# B&R Automation Studio project MotionTestBenchMaster (part 24)

#### MNM.sfc - Cyclic code
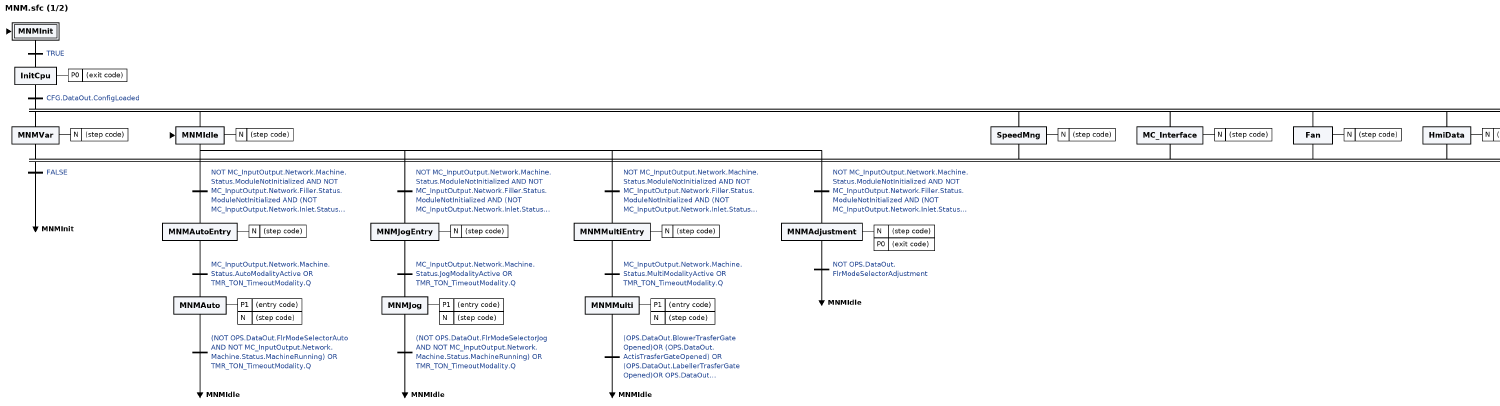
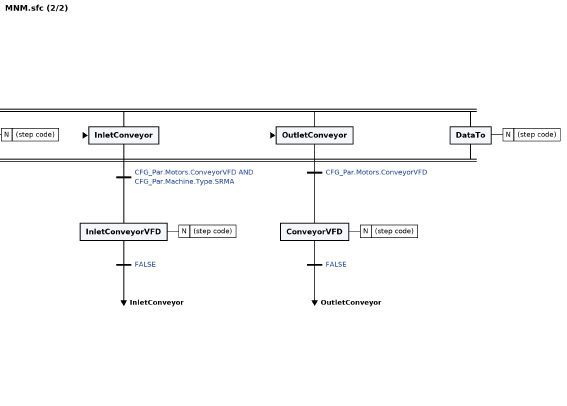
```iecst
PROGRAM _CYCLIC
INITIAL_STEP MNMInit:
END_STEP
TRANSITION FROM MNMInit TO InitCpu:=
TRUE
END_TRANSITION
STEP InitCpu:
END_STEP
EXIT_ACTION
InletConveyor_Hardware_CFG;
OutletConveyor_Hardware_CFG;
HMI_MNM_FlrSpeedWidget.AutoSpeedReq := REAL_TO_DINT(HMI_MNM_MinMachineSpeed);

HMI_CFG_PAR_1._020	:= TRUE;
HMI_CFG_PAR_1._160	:= _InCvrFC280.IN_ConfigPresent;//V 200.2.0
HMI_CFG_PAR_1._162	:= _OutCvrFC280.IN_ConfigPresent;

HMI_CFG_PAM_1._001	:= TRUE;//V 200.2.0
HMI_CFG_PAM_1._003	:= TRUE;
HMI_CFG_PAM_1._010	:= TRUE;
HMI_CFG_PAM_1._011	:= TRUE;
HMI_CFG_PAM_1._012	:= TRUE;
HMI_CFG_PAM_1._013	:= TRUE;
HMI_CFG_PAM_1._020	:= TRUE;

HMI_CFG_PAM_1._396	:= CFG_Par.Machine.Type.SRMA;//V 200.2.0
HMI_CFG_PAM_1._397	:= CFG_Par.Machine.Type.SRMA;//V 200.2.0
HMI_CFG_PAM_1._398	:= CFG_Par.Machine.Type.SRMA;//V 200.2.0
HMI_CFG_PAM_1._399	:= CFG_Par.Machine.Type.SRMA;//V 200.2.0
HMI_CFG_PAM_1._400	:= CFG_Par.Machine.Type.SRMA;//V 200.2.0
HMI_CFG_PAM_1._401	:= CFG_Par.Machine.Type.SRMA;//V 200.2.0
HMI_CFG_PAM_1._402	:= CFG_Par.Machine.Type.SRMA;//V 200.2.0
HMI_CFG_PAM_1._403	:= CFG_Par.Machine.Type.SRMA;//V 200.2.0
HMI_CFG_PAM_1._404	:= CFG_Par.ClosingUnit.Capper.Present;
HMI_CFG_PAM_1._405	:= CFG_Par.ClosingUnit.Capper.Present;
HMI_CFG_PAM_1._406	:= CFG_Par.ClosingUnit.Capper.Present;
HMI_CFG_PAM_1._407	:= CFG_Par.ClosingUnit.Capper.Present;
HMI_CFG_PAM_1._408	:= CFG_Par.ClosingUnit.Capper.Present;
HMI_CFG_PAM_1._409	:= CFG_Par.ClosingUnit.Capper.Present;
HMI_CFG_PAM_1._410	:= CFG_Par.ClosingUnit.Capper.Present;
HMI_CFG_PAM_1._411	:= CFG_Par.ClosingUnit.Capper.Present;
HMI_CFG_PAM_1._412	:= CFG_Par.Rinser.NoBottleNoSpray;//V 200.2.0
HMI_CFG_PAM_1._413	:= CFG_Par.Rinser.NoBottleNoSpray;//V 200.2.0
HMI_CFG_PAM_1._414	:= CFG_Par.Rinser.NoBottleNoSpray;//V 200.2.0
HMI_CFG_PAM_1._415	:= CFG_Par.Rinser.NoBottleNoSpray;//V 200.2.0
HMI_CFG_PAM_1._416	:= TRUE;//V 200.2.0
HMI_CFG_PAM_1._417	:= TRUE;//V 200.2.0
HMI_CFG_PAM_1._418	:= TRUE;//V 200.2.0
HMI_CFG_PAM_1._419	:= TRUE;//V 200.2.0
HMI_CFG_PAM_1._420	:= CFG_Par.ClosingUnit.Crowner.Present;
HMI_CFG_PAM_1._421	:= CFG_Par.ClosingUnit.Crowner.Present;
HMI_CFG_PAM_1._422	:= CFG_Par.ClosingUnit.Crowner.Present;
HMI_CFG_PAM_1._423	:= CFG_Par.ClosingUnit.Crowner.Present;
HMI_CFG_PAM_1._424	:= TRUE;
HMI_CFG_PAM_1._425	:= TRUE;
HMI_CFG_PAM_1._426	:= TRUE;
HMI_CFG_PAM_1._427	:= TRUE;
HMI_CFG_PAM_1._428	:= CFG_Par.FCI.Filltec OR CFG_Par.FCI.FTSystem OR CFG_Par.FCI.Heuft OR CFG_Par.FCI.Pressco OR CFG_Par.FCI.SIS OR CFG_Par.FCI.Stratec;//V4.A.A.1.7.0
HMI_CFG_PAM_1._429	:= CFG_Par.FCI.Filltec OR CFG_Par.FCI.FTSystem OR CFG_Par.FCI.Heuft OR CFG_Par.FCI.Pressco OR CFG_Par.FCI.SIS OR CFG_Par.FCI.Stratec;//V4.A.A.1.7.0
HMI_CFG_PAM_1._430	:= CFG_Par.FCI.Filltec OR CFG_Par.FCI.FTSystem OR CFG_Par.FCI.Heuft OR CFG_Par.FCI.Pressco OR CFG_Par.FCI.SIS OR CFG_Par.FCI.Stratec;//V4.A.A.1.7.0
HMI_CFG_PAM_1._431	:= CFG_Par.FCI.Filltec OR CFG_Par.FCI.FTSystem OR CFG_Par.FCI.Heuft OR CFG_Par.FCI.Pressco OR CFG_Par.FCI.SIS OR CFG_Par.FCI.Stratec;//V4.A.A.1.7.0
HMI_CFG_PAM_1._432	:= CFG_Par.FCI.Heuft OR CFG_Par.FCI.Stratec;
HMI_CFG_PAM_1._433	:= CFG_Par.FCI.Heuft OR CFG_Par.FCI.Stratec;
HMI_CFG_PAM_1._434	:= CFG_Par.FCI.Heuft OR CFG_Par.FCI.Stratec;
HMI_CFG_PAM_1._435	:= CFG_Par.FCI.Heuft OR CFG_Par.FCI.Stratec;
HMI_CFG_PAM_1._436	:= CFG_Par.Doser.Present; //v999hema
HMI_CFG_PAM_1._437	:= CFG_Par.Doser.Present; //v999hema
HMI_CFG_PAM_1._438	:= CFG_Par.Doser.Present; //v999hema
HMI_CFG_PAM_1._439	:= CFG_Par.Doser.Present; //v999hema

HMI_CFG_PAC_1._130	:= CFG_Par.Motors.FootbarPresent;
HMI_CFG_PAC_1._134  := CFG_Par.Machine.Type.SRMA AND CFG_Par.Lifting.Movements.Capper.UncoupledHeight > 0.0;//Capper Position For lifting movement
HMI_CFG_PAC_1._132	:= CFG_Par.Machine.Type.SRMA;
HMI_CFG_PAC_1._219	:= CFG_Par.Rinser.FootbarPresent;
HMI_CFG_PAC_1._220	:= CFG_Par.Rinser.FootbarPresent;
END_ACTION
TRANSITION FROM InitCpu TO (MNMVar,MNMIdle,SpeedMng,MC_Interface,Fan,HmiData,InletConveyor,OutletConveyor,DataTo):=
CFG.DataOut.ConfigLoaded
END_TRANSITION
STEP MNMVar:

VAR_MNM_NormalStop				:= AID.DataOut.ALR.Bit.ALR_MS_NormalStop;
VAR_MNM_QuickStop				:= AID.DataOut.ALR.Bit.ALR_MS_QuickStop;
VAR_MNM_NormalStopWithJog		:= AID.DataOut.ALR.Bit.ALR_MS_NormalWithJog;
VAR_MNM_NormalWithJogMnt		:= AID.DataOut.ALR.Bit.ALR_MS_NormalWithJogMnt; //V4.A.A.1.6.13
VAR_MNM_QuickStopWithJog		:= AID.DataOut.ALR.Bit.ALR_MS_QuickWithJog;
VAR_MNM_StopAfterEmpty 			:= AID.DataOut.ALR.Bit.ALR_CSR_StopAfterEmptying AND SFT.DataOut.MachineEmpty;//V 200.2.0

IF (MC_InputOutput.Network.Machine.Status.AutoModalityActive OR MC_InputOutput.Network.Machine.Status.MultiModalityActive) AND
	NOT VAR_MNM_NormalStop AND NOT VAR_MNM_QuickStop AND
	NOT VAR_MNM_NormalStopWithJog AND NOT  VAR_MNM_QuickStopWithJog AND NOT VAR_MNM_StopAfterEmpty THEN
	//added condition for stopping after pre-closing and washing cycle end//MasterBottle
	IF EDGEPOS(MAU_DumCon.DataOut.MachineStop) OR  EDGEPOS(SEL(CFG_Par.Process.BlendFill, SkdFlr.MachineStop, CrbFlr.MachineStop)) OR SFT.DataOut.FillingValvePositionReq OR CSR.DataOut.MachineStop OR EDGEPOS(CAP.DataOut.MachineStop) OR EDGEPOS(COP.DataOut.MachineStop) OR EDGEPOS(DOS.DataOut.MachineStop) OR EDGEPOS(RNS.DataOut.MachineStop) THEN//v999hema
		VAR_MNM_AutoStopRequest		:= TRUE;
		VAR_MNM_FlrAutoStopRequest	:= TRUE;
	END_IF

	IF (EDGEPOS(MAU_DumCon.DataOut.MachineStart) OR EDGEPOS(RNS.DataOut.MachineStart) OR EDGEPOS(SEL(CFG_Par.Process.BlendFill, SkdFlr.MachineStart, CrbFlr.MachineStart)) OR EDGEPOS(CAP.DataOut.MachineStart) OR EDGEPOS(COP.DataOut.MachineStart) OR EDGEPOS(DOS.DataOut.MachineStart) OR EDGEPOS(CRW.DataOut.MachineStart))
		AND NOT MAU_DumCon.DataOut.FillerReversePosReq AND NOT MAU_DumCon.DataOut.FillerFirstHalfPosReq AND NOT MAU_DumCon.DataOut.FillerSecondHalfPosReq THEN
		VAR_MNM_AutoStartRequest	:= TRUE;
		VAR_MNM_FlrAutoStartRequest := TRUE;
	END_IF
ELSE
	VAR_MNM_AutoStopRequest		:= FALSE;
	VAR_MNM_FlrAutoStopRequest	:= FALSE;
	VAR_MNM_AutoStartRequest	:= FALSE;
	VAR_MNM_FlrAutoStartRequest	:= FALSE;
END_IF

IF MC_InputOutput.Network.Machine.Status.AutoModalityActive THEN
	IF MC_InputOutput.Network.Machine.Status.MachineRunning THEN
		VAR_MNM_AutoStartRequest := FALSE;
	ELSE
		VAR_MNM_AutoStopRequest	:= FALSE;
	END_IF
	VAR_MNM_FlrAutoStopRequest	:= FALSE;
	VAR_MNM_FlrAutoStartRequest	:= FALSE;
ELSIF MC_InputOutput.Network.Machine.Status.MultiModalityActive THEN
	IF MC_InputOutput.Network.Filler.Status.ModuleRunning THEN
		VAR_MNM_FlrAutoStartRequest	:= FALSE;
	ELSE
		VAR_MNM_FlrAutoStopRequest	:= FALSE;
	END_IF
	VAR_MNM_AutoStopRequest		:= FALSE;
	VAR_MNM_AutoStartRequest	:= FALSE;
END_IF

(* Machine Start and Stop Management *)
VAR_MNM_FpMachineStartPb := EDGEPOS(HMI_CmdBar_PB[PB_FillerStartStop].Command);

//V4 200.2.0
VAR_MNM_MachineStart	:= IO_PB_FlStart.ON AND IO_PB_FlStart.Enable;
VAR_MNM_MachineStop		:= IO_PB_FlStop.ON;
END_STEP
STEP MNMIdle:
VAR_MNM_HornFlrRequest				:= FALSE;

MNM.DataOut.StartLightFixRequest	:= FALSE;
MNM.DataOut.StartLightBlinkRequest	:= FALSE;

TMR_TON_StartingHornElapsed.IN		:= FALSE;

TMR_TON_TimeoutModality.IN			:= FALSE;
TMR_TON_TimeoutModality();

FlrFmc.FillerOneStepReceived		:= FALSE;

MC_InputOutput.Network.Machine.Commands.MachineStart				:= FALSE;
MC_InputOutput.Network.Machine.Commands.JogPushButton				:= FALSE;
MC_InputOutput.Network.Machine.Commands.StepByStepModalityRequest	:= FALSE;
MC_InputOutput.Network.Machine.Commands.InMotionTimerModReq			:= FALSE;
MC_InputOutput.Network.Machine.Commands.StepByStepSingleAxisModReq	:= FALSE;//V1.7.2
MC_InputOutput.Network.Machine.Commands.PositioningModalityRequest	:= FALSE;//V1.7.2

MC_InputOutput.Network.Machine.Commands.AutoModalityRequest			:= FALSE;
MC_InputOutput.Network.Machine.Commands.AutoCombiModalityRequest	:= FALSE;
MC_InputOutput.Network.Machine.Commands.JogMachineModalityRequest	:= FALSE;
MC_InputOutput.Network.Machine.Commands.MultiModalityRequest		:= FALSE;

MC_InputOutput.Network.Filler.Commands.AutoFillerModule				:= FALSE;
MC_InputOutput.Network.Filler.Commands.JogFillerModule				:= FALSE;
MC_InputOutput.Network.Filler.Commands.StartFillerModule			:= FALSE;
MC_InputOutput.Network.Filler.Commands.JogPushButtonFillerModule	:= FALSE;

MC_InputOutput.Network.Inlet.Commands.AutoInletModule				:= FALSE;
MC_InputOutput.Network.Inlet.Commands.JogInletModule				:= FALSE;
MC_InputOutput.Network.Inlet.Commands.StartInletModule				:= FALSE;
MC_InputOutput.Network.Inlet.Commands.JogPushButtonInletModule		:= FALSE;

MC_InputOutput.Network.Outlet.Commands.AutoOutletModule				:= FALSE;
MC_InputOutput.Network.Outlet.Commands.JogOutletModule				:= FALSE;
MC_InputOutput.Network.Outlet.Commands.StartOutletModule			:= FALSE;
MC_InputOutput.Network.Outlet.Commands.JogPushButtonOutletModule	:= FALSE;
END_STEP
TRANSITION AutoMode FROM MNMIdle TO MNMAutoEntry:=
NOT MC_InputOutput.Network.Machine.Status.ModuleNotInitialized AND//v1.7.2a
NOT MC_InputOutput.Network.Filler.Status.ModuleNotInitialized AND//VXXXXXX
(NOT MC_InputOutput.Network.Inlet.Status.ModuleNotInitialized	OR MC_InputOutput.Network.Inlet.Status.ModuleReal)	AND
(NOT MC_InputOutput.Network.Outlet.Status.ModuleNotInitialized	OR MC_InputOutput.Network.Outlet.Status.ModuleReal)	AND
MC_InputOutput.Network.Machine.Status.EnableAuto				AND
OPS.DataOut.FlrModeSelectorAuto		AND //V4 200.2.0
NOT MC_InputOutput.Network.Machine.Exceptions.DcBusLowMachineException//V4.A.A.1.7.0
END_TRANSITION
TRANSITION JogMode FROM MNMIdle TO MNMJogEntry:=
NOT MC_InputOutput.Network.Machine.Status.ModuleNotInitialized AND//v1.7.2a
NOT MC_InputOutput.Network.Filler.Status.ModuleNotInitialized	AND
(NOT MC_InputOutput.Network.Inlet.Status.ModuleNotInitialized	OR MC_InputOutput.Network.Inlet.Status.ModuleReal)	AND
(NOT MC_InputOutput.Network.Outlet.Status.ModuleNotInitialized	OR MC_InputOutput.Network.Outlet.Status.ModuleReal)	AND
MC_InputOutput.Network.Machine.Status.EnableJog					AND
OPS.DataOut.FlrModeSelectorJog	AND
NOT MC_InputOutput.Network.Machine.Exceptions.DcBusLowMachineException//V4 200.2.0
END_TRANSITION
STEP MNMJogEntry:
MC_InputOutput.Network.Machine.Commands.JogMachineModalityRequest		:= TRUE;
TMR_TON_TimeoutModality(IN := TRUE, PT := t#2s);
END_STEP
TRANSITION JogModeActive FROM MNMJogEntry TO MNMJog:=
MC_InputOutput.Network.Machine.Status.JogModalityActive OR TMR_TON_TimeoutModality.Q
END_TRANSITION
STEP MNMJog:
MC_InputOutput.Network.Machine.Commands.JogMachineModalityRequest		:= TRUE;

IF VAR_MNM_NormalStop OR VAR_MNM_QuickStop THEN
	VAR_MNM_JogStep := MNM_JogFault;
ELSIF NOT (NOT MC_InputOutput.Network.Machine.Status.NoModalityActive AND MC_InputOutput.Network.Machine.Status.JogModalityActive) THEN
	VAR_MNM_JogStep := MNM_JogWaitStart;
ELSIF EDGENEG(OPS.DataOut.JogStartPb)  THEN
	VAR_MNM_JogStep := MNM_JogWaitStart;
END_IF

TMR_TON_StartingHornElapsed.IN	:= FALSE;
MC_InputOutput.Network.Machine.Commands.JogPushButton				:= FALSE;
VAR_MNM_HornFlrRequest	:= FALSE;

CASE VAR_MNM_JogStep OF
	MNM_JogWaitStart:
		IF OPS.DataOut.JogStartPb AND NOT CSR.DataOut.MachineStop THEN (*Master nuovo*)
			VAR_MNM_JogStep := MNM_JogHornBlow;
		END_IF

	MNM_JogHornBlow:
		TMR_TON_StartingHornElapsed.IN	:= TRUE;
		VAR_MNM_HornFlrRequest	:= TRUE;

		IF TMR_TON_StartingHornElapsed.Q THEN
			VAR_MNM_JogStep := MNM_JogMachineStart;
		END_IF

	MNM_JogMachineStart:
		MC_InputOutput.Network.Machine.Commands.JogPushButton := TRUE;

		IF MC_InputOutput.Network.Machine.Status.MachineRunning THEN
			VAR_MNM_JogStep := MNM_JogMachineRunning;
		END_IF

	MNM_JogMachineRunning:
		MC_InputOutput.Network.Machine.Commands.JogPushButton := TRUE;

	MNM_JogMachineStopping:
		IF NOT MC_InputOutput.Network.Machine.Status.MachineRunning THEN
			VAR_MNM_JogStep := MNM_JogWaitStart;
		END_IF

	MNM_JogFault:
		IF NOT VAR_MNM_NormalStop AND NOT VAR_MNM_QuickStop THEN
			VAR_MNM_JogStep := MNM_JogWaitStart;
		END_IF
END_CASE

TMR_TON_StartingHornElapsed(PT:= t#2s);
END_STEP
ENTRY_ACTION
VAR_MNM_JogStep := MNM_JogWaitStart;
END_ACTION
TRANSITION IdleMode FROM MNMJog TO MNMIdle:=
(NOT OPS.DataOut.FlrModeSelectorJog AND NOT MC_InputOutput.Network.Machine.Status.MachineRunning) OR //V 200.2.0
TMR_TON_TimeoutModality.Q
END_TRANSITION
(* @SFCISJUMP := 'MNMIdle' *)
TRANSITION MultiMode FROM MNMIdle TO MNMMultiEntry:=
NOT MC_InputOutput.Network.Machine.Status.ModuleNotInitialized AND
NOT MC_InputOutput.Network.Filler.Status.ModuleNotInitialized	AND
(NOT MC_InputOutput.Network.Inlet.Status.ModuleNotInitialized	OR MC_InputOutput.Network.Inlet.Status.ModuleReal)	AND
(NOT MC_InputOutput.Network.Outlet.Status.ModuleNotInitialized	OR MC_InputOutput.Network.Outlet.Status.ModuleReal)	AND
NOT OPS.DataOut.FlrModeSelectorAdjustment	AND
MC_InputOutput.Network.Machine.Status.EnableMulti	AND
NOT (OPS.DataOut.BlowerTrasferGateOpened AND OPS.DataOut.ActisTrasferGateOpened)AND //da cambiare
NOT MC_InputOutput.Network.Machine.Exceptions.DcBusLowMachineException
END_TRANSITION
STEP MNMMultiEntry:
MC_InputOutput.Network.Machine.Commands.MultiModalityRequest	:= TRUE;
TMR_TON_TimeoutModality(IN := TRUE, PT := t#2s);
END_STEP
TRANSITION MultiModeActive FROM MNMMultiEntry TO MNMMulti:=
MC_InputOutput.Network.Machine.Status.MultiModalityActive OR TMR_TON_TimeoutModality.Q
END_TRANSITION
STEP MNMMulti:
MC_InputOutput.Network.Machine.Commands.MultiModalityRequest	:= TRUE;

(* FILLER MULTI *)
IF EDGE(OPS.DataOut.FlrModeSelectorAuto) THEN
	VAR_MNM_FlrMultiStep := MNM_MultiModeSelection;
ELSIF VAR_MNM_FlrMultiStep >= MNM_MultiAutoWaitStart AND VAR_MNM_FlrMultiStep <= MNM_MultiAutoMachineStopping THEN
	IF VAR_MNM_NormalStop OR VAR_MNM_QuickStop OR VAR_MNM_NormalStopWithJog OR VAR_MNM_QuickStopWithJog OR VAR_MNM_StopAfterEmpty OR VAR_MNM_StopIfNotEmpty THEN
		VAR_MNM_FlrMultiStep := MNM_MultiFault;
	ELSIF NOT VAR_MNM_MachineStop OR VAR_MNM_FlrAutoStopRequest THEN
		VAR_MNM_FlrMultiStep := MNM_MultiAutoMachineStopping;
	END_IF
ELSIF VAR_MNM_FlrMultiStep >= MNM_MultiJogWaitStart AND VAR_MNM_FlrMultiStep <= MNM_MultiJogMachineStopping THEN
	IF VAR_MNM_NormalStop OR VAR_MNM_QuickStop THEN
		VAR_MNM_FlrMultiStep := MNM_MultiFault;
	ELSIF EDGENEG(OPS.DataOut.JogStartPb)  THEN
		VAR_MNM_FlrMultiStep := MNM_MultiJogMachineStopping;
	END_IF
END_IF

TMR_TON_StartingHornElapsed.IN	:= FALSE;
MC_InputOutput.Network.Filler.Commands.AutoFillerModule				:= FALSE;
MC_InputOutput.Network.Filler.Commands.StartFillerModule			:= FALSE;
MC_InputOutput.Network.Filler.Commands.JogFillerModule				:= FALSE;
MC_InputOutput.Network.Filler.Commands.JogPushButtonFillerModule	:= FALSE;
VAR_MNM_HornFlrRequest					:= FALSE;
MNM.DataOut.StartLightFixRequest		:= FALSE;
MNM.DataOut.StartLightBlinkRequest		:= FALSE;

CASE VAR_MNM_FlrMultiStep OF
	MNM_MultiModeSelection:
		IF OPS.DataOut.FlrModeSelectorAuto AND MC_InputOutput.Network.Filler.Status.EnableAutoModality THEN
			VAR_MNM_FlrMultiStep := MNM_MultiAutoWaitStart;
		ELSIF OPS.DataOut.FlrModeSelectorJog AND MC_InputOutput.Network.Filler.Status.EnableJogModality THEN
			VAR_MNM_FlrMultiStep := MNM_MultiJogWaitStart;
		END_IF

	MNM_MultiAutoWaitStart:
		MC_InputOutput.Network.Filler.Commands.AutoFillerModule := TRUE;
		MNM.DataOut.StartLightBlinkRequest	:= TRUE;

		IF ((VAR_MNM_MachineStart OR VAR_MNM_FlrAutoStartRequest) AND VAR_MNM_MachineStop AND MC_InputOutput.Network.Filler.Status.EnableAutoModality) THEN
			VAR_MNM_FlrMultiStep	:= MNM_MultiAutoHornBlow;
		ELSIF VAR_MNM_AutoVortexCalibActive THEN
			VAR_MNM_FlrMultiStep	:= MNM_MultiVortexCalibIdle;
		ELSIF FmcFlr.VortexCalibrActive THEN
			VAR_MNM_FlrMultiStep 	:= MNM_MultiVortexCalibHornBlow;
		ELSIF HMI_MNM_PB[PB_MNM_AxisStepByStep].ON THEN
			VAR_MNM_FlrMultiStep 	:= MNM_MultiStepHornBlow;
		ELSIF HMI_MNM_PB[PB_MNM_FootboardPosition].ON THEN
			VAR_MNM_FlrMultiStep 	:= MNM_MultiFootboardHornBlow;
		ELSIF CAP.DataOut.GreasingPositioningReq OR CSR.DataOut.CapPositioningReq THEN//V4.A.A.1.7.0
			VAR_MNM_FlrMultiStep	:= MNM_MultiCapperPosHornBlow;
		END_IF

	MNM_MultiAutoHornBlow:
		MC_InputOutput.Network.Filler.Commands.AutoFillerModule	:= TRUE;
		MNM.DataOut.StartLightFixRequest	:= TRUE;
		TMR_TON_StartingHornElapsed.IN		:= TRUE;
		VAR_MNM_HornFlrRequest	:= TRUE;

		IF NOT ((VAR_MNM_MachineStart OR VAR_MNM_FlrAutoStartRequest) AND VAR_MNM_MachineStop AND MC_InputOutput.Network.Filler.Status.EnableAutoModality) THEN
			VAR_MNM_FlrMultiStep := MNM_MultiAutoWaitStart;
		END_IF

		IF TMR_TON_StartingHornElapsed.Q THEN
			VAR_MNM_FlrMultiStep := MNM_MultiAutoMachineStart;
		END_IF

	MNM_MultiAutoMachineStart:
		MC_InputOutput.Network.Filler.Commands.AutoFillerModule		:= TRUE;
		MC_InputOutput.Network.Filler.Commands.StartFillerModule	:= TRUE;
		MNM.DataOut.StartLightFixRequest	:= TRUE;

		IF MC_InputOutput.Network.Filler.Status.ModuleRunning THEN
			VAR_MNM_FlrMultiStep := MNM_MultiAutoMachineRunning;
		END_IF

	MNM_MultiAutoMachineRunning:	//Wait stop PB or Fault
		MC_InputOutput.Network.Filler.Commands.AutoFillerModule		:= TRUE;
		MC_InputOutput.Network.Filler.Commands.StartFillerModule	:= TRUE;
		MNM.DataOut.StartLightFixRequest	:= TRUE;

	MNM_MultiAutoMachineStopping:
		MC_InputOutput.Network.Filler.Commands.AutoFillerModule		:= TRUE;

		IF NOT MC_InputOutput.Network.Filler.Status.ModuleRunning THEN
			VAR_MNM_FlrMultiStep := MNM_MultiAutoWaitStart;
		END_IF

	MNM_MultiVortexCalibHornBlow:
		TMR_TON_StartingHornElapsed.IN	:= TRUE;
		VAR_MNM_HornFlrRequest	:= TRUE;

		IF TMR_TON_StartingHornElapsed.Q THEN
			VAR_MNM_FlrMultiStep := MNM_MultiVortexCalibPosStart;
		END_IF

	MNM_MultiVortexCalibPosStart:
		MC_InputOutput.Network.Filler.Parameters.StepNumber	:= 1;
		MC_InputOutput.Network.Filler.Commands.StepByStepModalityRequest	:= TRUE;

		IF MC_InputOutput.Network.Filler.Status.StepByStepModalityActive THEN
			VAR_MNM_FlrMultiStep := MNM_MultiVortexCalibPosWaitStop;
		END_IF

	MNM_MultiVortexCalibPosWaitStop:
		IF NOT MC_InputOutput.Network.Filler.Status.StepByStepModalityActive AND NOT MC_InputOutput.Network.Filler.Status.ModuleRunning THEN
			VAR_MNM_FlrMultiStep := MNM_MultiVortexCalibIdle;
			VAR_MNM_AutoVortexCalibActive := TRUE;
		END_IF

	MNM_MultiVortexCalibIdle:
		IF EDGEPOS(FmcFlr.FillerOneStepReq) THEN
			VAR_MNM_FlrMultiStep := MNM_MultiStepFmcHornBlow;
		END_IF

		IF NOT FmcFlr.VortexCalibrActive THEN
			VAR_MNM_AutoVortexCalibActive := FALSE;
			VAR_MNM_FlrMultiStep := MNM_MultiAutoWaitStart;
		END_IF

	MNM_MultiStepFmcHornBlow:
		TMR_TON_StartingHornElapsed.IN	:= TRUE;
		VAR_MNM_HornFlrRequest	:= TRUE;

		IF TMR_TON_StartingHornElapsed.Q THEN
			FlrFmc.FillerOneStepReceived	:= FmcFlr.FillerOneStepReq;
			VAR_MNM_FlrMultiStep := MNM_MultiStepFmcStart;
		END_IF

	MNM_MultiStepFmcStart:
		MC_InputOutput.Network.Filler.Parameters.StepNumber	:= 1;
		MC_InputOutput.Network.Filler.Commands.StepByStepModalityRequest	:= TRUE;

		IF MC_InputOutput.Network.Filler.Status.StepByStepModalityActive THEN
			VAR_MNM_FlrMultiStep := MNM_MultiStepFmcWaitStop;
		END_IF

	MNM_MultiStepFmcWaitStop:
		IF NOT MC_InputOutput.Network.Filler.Status.StepByStepModalityActive AND NOT MC_InputOutput.Network.Filler.Status.ModuleRunning THEN
			VAR_MNM_FlrMultiStep := MNM_MultiVortexCalibIdle;
		END_IF

	MNM_MultiStepHornBlow:
		TMR_TON_StartingHornElapsed.IN	:= TRUE;
		VAR_MNM_HornFlrRequest	:= TRUE;

		IF TMR_TON_StartingHornElapsed.Q THEN
			VAR_MNM_FlrMultiStep := MNM_MultiStepStart;
		END_IF

	MNM_MultiStepStart:
		MC_InputOutput.Network.Filler.Parameters.StepNumber	:= HMI_MNM_AxisStepByStepOffset;
		MC_InputOutput.Network.Filler.Commands.StepByStepModalityRequest	:= TRUE;

		IF MC_InputOutput.Network.Filler.Status.StepByStepModalityActive THEN
			VAR_MNM_FlrMultiStep := MNM_MultiStepWaitStop;
		END_IF

	MNM_MultiStepWaitStop:
		IF NOT MC_InputOutput.Network.Filler.Status.StepByStepModalityActive AND NOT MC_InputOutput.Network.Filler.Status.ModuleRunning THEN
			VAR_MNM_FlrMultiStep := MNM_MultiAutoWaitStart;
		END_IF

	MNM_MultiFootboardHornBlow:
		TMR_TON_StartingHornElapsed.IN	:= TRUE;
		VAR_MNM_HornFlrRequest	:= TRUE;

		IF TMR_TON_StartingHornElapsed.Q THEN
			VAR_MNM_FlrMultiStep := MNM_MultiFootboardStart;
		END_IF

	MNM_MultiFootboardStart:
		IF LREAL_TO_INT(MC_InputOutput.Network.Filler.Status.FillerAbsolutePosition / 360.0) < HMI_PAC_1._130 THEN
			MC_InputOutput.Network.Filler.Parameters.StepNumber		:= HMI_PAC_1._130 - (LREAL_TO_INT(MC_InputOutput.Network.Filler.Status.FillerAbsolutePosition / 360.0));
		ELSE
			MC_InputOutput.Network.Filler.Parameters.StepNumber	:= HMI_PAC_1._100 - (LREAL_TO_INT(MC_InputOutput.Network.Filler.Status.FillerAbsolutePosition / 360.0)) + HMI_PAC_1._130;
		END_IF

		MC_InputOutput.Network.Filler.Commands.StepByStepModalityRequest	:= TRUE;

		IF MC_InputOutput.Network.Filler.Status.StepByStepModalityActive THEN
			VAR_MNM_FlrMultiStep := MNM_MultiFootboardWaitStop;
		END_IF

	MNM_MultiFootboardWaitStop:
		IF NOT MC_InputOutput.Network.Filler.Status.StepByStepModalityActive AND NOT MC_InputOutput.Network.Filler.Status.ModuleRunning THEN
			VAR_MNM_FlrMultiStep := MNM_MultiAutoWaitStart;
		END_IF

	MNM_MultiCapperPosHornBlow:

	MNM_MultiCapperPosStart:

	MNM_MultiCapperPosWaitStop:

	MNM_MultiCapperFinePosStart:

	MNM_MultiCapperFinePosWaitStop:

	MNM_MultiJogWaitStart:
		MC_InputOutput.Network.Filler.Commands.JogFillerModule	:= TRUE;
		IF OPS.DataOut.JogStartPb THEN
			VAR_MNM_FlrMultiStep := MNM_MultiJogHornBlow;
		END_IF

	MNM_MultiJogHornBlow:
		MC_InputOutput.Network.Filler.Commands.JogFillerModule	:= TRUE;
		TMR_TON_StartingHornElapsed.IN	:= TRUE;
		VAR_MNM_HornFlrRequest	:= TRUE;

		IF TMR_TON_StartingHornElapsed.Q THEN
			VAR_MNM_FlrMultiStep := MNM_MultiJogMachineStart;
		END_IF

	MNM_MultiJogMachineStart:
		MC_InputOutput.Network.Filler.Commands.JogFillerModule	:= TRUE;
		MC_InputOutput.Network.Filler.Commands.JogPushButtonFillerModule := TRUE;

		IF MC_InputOutput.Network.Filler.Status.ModuleRunning THEN
			VAR_MNM_FlrMultiStep := MNM_MultiJogMachineRunning;
		END_IF

	MNM_MultiJogMachineRunning:
		MC_InputOutput.Network.Filler.Commands.JogFillerModule	:= TRUE;
		MC_InputOutput.Network.Filler.Commands.JogPushButtonFillerModule:= TRUE;

	MNM_MultiJogMachineStopping:
		MC_InputOutput.Network.Filler.Commands.JogFillerModule	:= TRUE;
		IF NOT MC_InputOutput.Network.Filler.Status.ModuleRunning THEN
			VAR_MNM_FlrMultiStep := MNM_MultiJogWaitStart;
		END_IF

	MNM_MultiFault:
		MC_InputOutput.Network.Filler.Commands.AutoFillerModule		:= OPS.DataOut.FlrModeSelectorAuto AND MC_InputOutput.Network.Filler.Status.EnableAutoModality;//V4.A.A.1.6.12d
		MC_InputOutput.Network.Filler.Commands.JogFillerModule		:= OPS.DataOut.FlrModeSelectorJog AND MC_InputOutput.Network.Filler.Status.EnableJogModality;//V4.A.A.1.6.12d

		IF NOT (VAR_MNM_NormalStop OR VAR_MNM_QuickStop OR VAR_MNM_NormalStopWithJog OR VAR_MNM_QuickStopWithJog OR VAR_MNM_StopAfterEmpty OR VAR_MNM_StopIfNotEmpty) THEN
			VAR_MNM_FlrMultiStep := MNM_MultiAutoWaitStart;//V4.A.A.1.6.12d
		ELSIF MC_InputOutput.Network.Filler.Status.ModuleJogActive THEN
			IF NOT VAR_MNM_NormalStop AND NOT VAR_MNM_QuickStop THEN
				VAR_MNM_FlrMultiStep := MNM_MultiJogWaitStart;
			END_IF
		END_IF
END_CASE

TMR_TON_StartingHornElapsed(PT:= t#2s);
END_STEP
ENTRY_ACTION
VAR_MNM_FlrMultiStep		:= MNM_MultiModeSelection;
VAR_MNM_FlrInletMultiStep	:= MNM_MultiModeSelection;
END_ACTION
TRANSITION IdleMode FROM MNMMulti TO MNMIdle:=
(OPS.DataOut.BlowerTrasferGateOpened)OR//da controllare in collaudo
(OPS.DataOut.ActisTrasferGateOpened) OR//da controllare in collaudo
(OPS.DataOut.LabellerTrasferGateOpened)OR//da controllare in collaudo
OPS.DataOut.FlrModeSelectorAdjustment OR TMR_TON_TimeoutModality.Q
END_TRANSITION
(* @SFCISJUMP := 'MNMIdle' *)
TRANSITION AdjustmentMode FROM MNMIdle TO MNMAdjustment:=
NOT MC_InputOutput.Network.Machine.Status.ModuleNotInitialized AND
NOT MC_InputOutput.Network.Filler.Status.ModuleNotInitialized	AND
(NOT MC_InputOutput.Network.Inlet.Status.ModuleNotInitialized	OR MC_InputOutput.Network.Inlet.Status.ModuleReal)	AND
(NOT MC_InputOutput.Network.Outlet.Status.ModuleNotInitialized	OR MC_InputOutput.Network.Outlet.Status.ModuleReal)	AND
OPS.DataOut.FlrModeSelectorAdjustment AND
NOT MC_InputOutput.Network.Machine.Exceptions.DcBusLowMachineException
END_TRANSITION
STEP MNMAdjustment:
IF VAR_MNM_NormalStop OR VAR_MNM_QuickStop OR VAR_MNM_NormalStopWithJog OR VAR_MNM_QuickStopWithJog OR VAR_MNM_StopAfterEmpty OR VAR_MNM_StopIfNotEmpty THEN//V4.A.A.1.7.0
	VAR_MNM_AdjustmentStep := MNM_AdjFault;
END_IF
IF EDGEPOS(HMI_MNM_PB[PB_MNM_AxisPositioning].ON) THEN
	MC_InputOutput.Network.Machine.Commands.PositioningModalityRequest	:=  TRUE;
ELSIF MC_InputOutput.Network.Machine.Status.PositioningModalityActive OR NOT HMI_MNM_PB[PB_MNM_AxisPositioning].ON THEN
	MC_InputOutput.Network.Machine.Commands.PositioningModalityRequest	:=  FALSE;
END_IF

IF EDGENEG(MC_InputOutput.Network.Machine.Status.PositioningModalityActive) THEN
	HMI_MNM_AxisPositionOffset	:= 0.0;
END_IF

IF EDGEPOS(HMI_MNM_PB[PB_MNM_AxisHoming].ON) THEN
	MC_InputOutput.Network.Machine.Commands.SelectiveHomeModalityRequest	:= TRUE;
ELSIF MC_InputOutput.Network.Machine.Status.SelectiveHomeModalityActive OR NOT HMI_MNM_PB[PB_MNM_AxisHoming].ON THEN
	MC_InputOutput.Network.Machine.Commands.SelectiveHomeModalityRequest	:= FALSE;
END_IF

MC_InputOutput.Network.Machine.Commands.BrakeReleaseModalityRequest	:= HMI_MNM_PB[PB_MNM_BrakeRelease].ON;

MC_InputOutput.Network.Machine.Commands.VelocityModalityRequest		:= HMI_MNM_PB[PB_MNM_VelocityTest].ON;
MC_InputOutput.Network.Machine.Parameters.ManualVelocity			:= REAL_TO_UINT(HMI_MNM_ConveyorSpeed / 10.0);

TMR_TON_StartingHornElapsed.IN	:= FALSE;
VAR_MNM_HornFlrRequest	:= FALSE;
MNM.DataOut.StartLightFixRequest	:= FALSE;
MNM.DataOut.StartLightBlinkRequest	:= FALSE;

CASE VAR_MNM_AdjustmentStep OF
	MNM_AdjWaitStart:
		VAR_MNM_AdjAxisPositionOffset := 0.0;

		//MNM.DataOut.StartLightBlinkRequest	:= TRUE; v4 200.2.0 // no blink PB start in Adjustment modality

		IF HMI_MNM_PB[PB_MNM_FootboardPosition].ON THEN
			VAR_MNM_AdjustmentStep := MNM_AdjFillerFootbarSettingPos;
		ELSIF  HMI_MNM_PB[PB_MNM_RinserFootboardPosition].ON THEN
			VAR_MNM_AdjustmentStep := MNM_AdjRinserFootbarSettingPos;
		ELSIF CAP.DataOut.GreasingPositioningReq  THEN
			VAR_MNM_AdjustmentStep := MNM_AdjCapGreasingSettingPos;
		ELSIF CSR.DataOut.CrwPositioningReq THEN
			VAR_MNM_AdjustmentStep := MNM_AdjCrownerSettingPos;
		ELSIF CSR.DataOut.CapPositioningReq THEN
			VAR_MNM_AdjustmentStep := MNM_AdjCapperSettingPos;
		END_IF
	//Filler Footbar
	MNM_AdjFillerFootbarSettingPos:

		VAR_MNM_AdjAxisFillerFootBar := TRUE;

		HMI_MNM_AxisSelected := CFG_MC.Mechanical.ReferenceId.Filler + CST_FillerSubModuleHmiStart;
		VAR_MNM_AdjAxisPositionOffset := 0.0;

		IF LREAL_TO_INT(MC_InputOutput.Network.Filler.Status.FillerAbsolutePosition / 360.0) < HMI_PAC_1._130 THEN
			MC_InputOutput.Network.Machine.Parameters.StepNumber		:= HMI_PAC_1._130 - (LREAL_TO_INT(MC_InputOutput.Network.Filler.Status.FillerAbsolutePosition / 360.0));
		ELSE
			MC_InputOutput.Network.Machine.Parameters.StepNumber	:= HMI_PAC_1._100 - (LREAL_TO_INT(MC_InputOutput.Network.Filler.Status.FillerAbsolutePosition / 360.0)) + HMI_PAC_1._130;
		END_IF

		VAR_MNM_AdjustmentStep := MNM_AdjHornBlow;
	//Rinser Footbar
	MNM_AdjRinserFootbarSettingPos:

		VAR_MNM_AdjAxisRinserFootBar	:= TRUE;

		HMI_MNM_AxisSelected := CFG_MC.Mechanical.ReferenceId.Rinser + CST_FillerSubModuleHmiStart;
		VAR_MNM_AdjAxisPositionOffset := 0.0;

		IF LREAL_TO_INT(MC_InputOutput.Network.Filler.Status.RinserAbsolutePosition / 360.0) < HMI_PAC_1._220 THEN
			MC_InputOutput.Network.Machine.Parameters.StepNumber		:= HMI_PAC_1._220 - (LREAL_TO_INT(MC_InputOutput.Network.Filler.Status.RinserAbsolutePosition / 360.0));
		ELSE
			MC_InputOutput.Network.Machine.Parameters.StepNumber	:= HMI_PAC_1._200- (LREAL_TO_INT(MC_InputOutput.Network.Filler.Status.RinserAbsolutePosition / 360.0)) + HMI_PAC_1._220;
		END_IF

		VAR_MNM_AdjustmentStep := MNM_AdjHornBlow;
	//Doser Pos
	MNM_AdjDoserFootbarSettingPos:

		HMI_MNM_AxisSelected := CFG_MC.Mechanical.ReferenceId.Rinser + CST_FillerSubModuleHmiStart;
		VAR_MNM_AdjAxisPositionOffset := 0.0;

		IF LREAL_TO_INT(MC_InputOutput.Network.Filler.Status.FillerAbsolutePosition / 360.0) < HMI_PAC_1._130 THEN//
			MC_InputOutput.Network.Machine.Parameters.StepNumber		:= HMI_PAC_1._130 - (LREAL_TO_INT(MC_InputOutput.Network.Filler.Status.FillerAbsolutePosition / 360.0));
		ELSE
			MC_InputOutput.Network.Machine.Parameters.StepNumber	:= HMI_PAC_1._500- (LREAL_TO_INT(MC_InputOutput.Network.Filler.Status.FillerAbsolutePosition / 360.0)) + HMI_PAC_1._130;
		END_IF

		VAR_MNM_AdjustmentStep := MNM_AdjHornBlow;
	//Capper pos For lifting
	MNM_AdjCapperSettingPos:

		HMI_MNM_AxisSelected := CFG_MC.Mechanical.ReferenceId.Capper + CST_FillerSubModuleHmiStart;
		VAR_MNM_AdjAxisPositionOffset := HMI_PAM_3._540;

		IF LREAL_TO_INT(MC_InputOutput.Network.Filler.Status.CapperAbsolutePosition / 360.0) < HMI_PAC_1._134 THEN
			MC_InputOutput.Network.Machine.Parameters.StepNumber		:= HMI_PAC_1._134 - (LREAL_TO_INT(MC_InputOutput.Network.Filler.Status.CapperAbsolutePosition / 360.0));//Fra
		ELSE
			MC_InputOutput.Network.Machine.Parameters.StepNumber	:= HMI_PAC_1._400 - (LREAL_TO_INT(MC_InputOutput.Network.Filler.Status.CapperAbsolutePosition / 360.0)) + HMI_PAC_1._134;//Fra
		END_IF

		VAR_MNM_AdjustmentStep := MNM_AdjHornBlow;

	//Crowner  Pos For Lifting
	MNM_AdjCrownerSettingPos:

		HMI_MNM_AxisSelected := CFG_MC.Mechanical.ReferenceId.Crowner + CST_FillerSubModuleHmiStart;
		VAR_MNM_AdjAxisPositionOffset := HMI_PAM_3._410;

		IF LREAL_TO_INT(MC_InputOutput.Network.Filler.Status.CrownerAbsolutePosition / 360.0) < HMI_PAC_1._133 THEN
			MC_InputOutput.Network.Machine.Parameters.StepNumber		:= HMI_PAC_1._133 - (LREAL_TO_INT(MC_InputOutput.Network.Filler.Status.CrownerAbsolutePosition / 360.0));//Fra
		ELSE
			MC_InputOutput.Network.Machine.Parameters.StepNumber	:= HMI_PAC_1._300 - (LREAL_TO_INT(MC_InputOutput.Network.Filler.Status.CrownerAbsolutePosition / 360.0)) + HMI_PAC_1._133;//Fra
		END_IF

		VAR_MNM_AdjustmentStep := MNM_AdjHornBlow;
	//Capper Greasing Pos
	MNM_AdjCapGreasingSettingPos:

		HMI_MNM_AxisSelected := CFG_MC.Mechanical.ReferenceId.Capper + CST_FillerSubModuleHmiStart;
		VAR_MNM_AdjAxisPositionOffset := HMI_PAM_3._528;

		IF LREAL_TO_INT(MC_InputOutput.Network.Filler.Status.CapperAbsolutePosition / 360.0) < HMI_PAC_1._130 THEN
			MC_InputOutput.Network.Machine.Parameters.StepNumber		:= HMI_PAC_1._131 - (LREAL_TO_INT(MC_InputOutput.Network.Filler.Status.CapperAbsolutePosition / 360.0));//Fra
		ELSE
			MC_InputOutput.Network.Machine.Parameters.StepNumber	:= HMI_PAC_1._400 - (LREAL_TO_INT(MC_InputOutput.Network.Filler.Status.CapperAbsolutePosition / 360.0)) + HMI_PAC_1._131;//FRa
		END_IF

		VAR_MNM_AdjustmentStep := MNM_AdjHornBlow;

	MNM_AdjHornBlow:

		TMR_TON_StartingHornElapsed.IN	:= TRUE;
		VAR_MNM_HornFlrRequest	:= TRUE;

		IF TMR_TON_StartingHornElapsed.Q THEN
			VAR_MNM_AdjustmentStep := MNM_AdjAxisStart;
		END_IF

	MNM_AdjAxisStart:

		MC_InputOutput.Network.Machine.Commands.StepByStepSingleAxisModReq := TRUE;

		IF MC_InputOutput.Network.Machine.Status.StepByStepSingleAxisModeActive THEN
			VAR_MNM_AdjustmentStep := MNM_AdjAxisWaitStop;
		END_IF

	MNM_AdjAxisWaitStop:

		VAR_MNM_AdjAxisFillerFootBar	:= FALSE; //V4.A.A.1.7.0
		VAR_MNM_AdjAxisRinserFootBar	:= FALSE; //V4.A.A.1.7.0

		MC_InputOutput.Network.Machine.Commands.StepByStepSingleAxisModReq := FALSE;

		IF NOT MC_InputOutput.Network.Machine.Status.StepByStepSingleAxisModeActive AND NOT MC_InputOutput.Network.Machine.Status.MachineRunning THEN
			IF VAR_MNM_AdjAxisPositionOffset <> 0.0 THEN
				VAR_MNM_AdjustmentStep := MNM_AdjAxisPosStart;
			ELSE
				VAR_MNM_AdjustmentStep := MNM_AdjAxisStopped;
			END_IF
		END_IF

	MNM_AdjAxisPosStart:
		HMI_MNM_AxisPositionOffset := VAR_MNM_AdjAxisPositionOffset;
		MC_InputOutput.Network.Machine.Commands.PositioningModalityRequest := TRUE;

		IF MC_InputOutput.Network.Machine.Status.PositioningModalityActive THEN
			MC_InputOutput.Network.Machine.Commands.PositioningModalityRequest	:= FALSE;
			VAR_MNM_AdjustmentStep := MNM_AdjAxisPosWaitStop;
		END_IF

	MNM_AdjAxisPosWaitStop:
		MC_InputOutput.Network.Machine.Commands.PositioningModalityRequest			:= FALSE;
		IF NOT MC_InputOutput.Network.Machine.Status.PositioningModalityActive AND NOT MC_InputOutput.Network.Machine.Status.MachineRunning THEN
			MNM.DataOut.SingleAxisInPosition	:= TRUE;
			MNM.DataOut.CapperPositioningDone	:= TRUE;//v4.A.A.1.7.0
			VAR_MNM_AdjustmentStep := MNM_AdjAxisStopped;
		END_IF

	MNM_AdjAxisStopped:

		MNM.DataOut.SingleAxisInPosition	:= TRUE;
		MNM.DataOut.CapperPositioningDone	:= TRUE;//v4.A.A.1.7.0

		IF NOT CAP.DataOut.GreasingPositioningReq AND NOT CSR.DataOut.CapPositioningReq AND NOT CSR.DataOut.CrwPositioningReq  THEN
			MNM.DataOut.SingleAxisInPosition	:= FALSE;
			MNM.DataOut.CapperPositioningDone	:= FALSE;//v4.A.A.1.7.0
			VAR_MNM_AdjustmentStep := MNM_AdjWaitStart;
		END_IF

	MNM_AdjFault:
		MC_InputOutput.Network.Machine.Commands.PositioningModalityRequest := FALSE;
		MC_InputOutput.Network.Machine.Commands.StepByStepSingleAxisModReq := FALSE;

		IF NOT MC_InputOutput.Network.Machine.Status.StepByStepModalityActive AND NOT MC_InputOutput.Network.Machine.Status.MachineRunning AND
			NOT MC_InputOutput.Network.Machine.Status.PositioningModalityActive THEN
			VAR_MNM_AdjustmentStep := MNM_AdjWaitStart;
		END_IF
END_CASE

TMR_TON_StartingHornElapsed(PT:= t#2s);
END_STEP
EXIT_ACTION
VAR_MNM_AdjAxisFillerFootBar		:= FALSE;//V1.7.2
VAR_MNM_AdjAxisRinserFootBar		:= FALSE;//V1.7.2
MNM.DataOut.SingleAxisInPosition	:= FALSE;//V1.7.2
MNM.DataOut.CapperPositioningDone	:= FALSE;//V1.7.2
END_ACTION
TRANSITION IdleMode FROM MNMAdjustment TO MNMIdle:=
NOT OPS.DataOut.FlrModeSelectorAdjustment
END_TRANSITION
(* @SFCISJUMP := 'MNMIdle' *)
STEP MNMAutoEntry:
MC_InputOutput.Network.Machine.Commands.AutoModalityRequest	:= TRUE;
TMR_TON_TimeoutModality(IN := TRUE, PT := t#2s);
END_STEP
TRANSITION AutoModeActive FROM MNMAutoEntry TO MNMAuto:=
MC_InputOutput.Network.Machine.Status.AutoModalityActive OR TMR_TON_TimeoutModality.Q
END_TRANSITION
STEP MNMAuto:
MC_InputOutput.Network.Machine.Commands.AutoModalityRequest	:= TRUE;

IF VAR_MNM_NormalStop OR VAR_MNM_QuickStop OR VAR_MNM_NormalStopWithJog OR VAR_MNM_QuickStopWithJog OR VAR_MNM_StopAfterEmpty OR VAR_MNM_StopIfNotEmpty THEN
	VAR_MNM_AutoStep := MNM_AutoFault;
ELSIF NOT (NOT MC_InputOutput.Network.Machine.Status.NoModalityActive AND (MC_InputOutput.Network.Machine.Status.AutoModalityActive OR
	MC_InputOutput.Network.Machine.Status.StepByStepModalityActive  OR
	MC_InputOutput.Network.Machine.Status.StepByStepSingleAxisModeActive OR MC_InputOutput.Network.Machine.Status.StepByStepSingleAxisRevModActive )) AND NOT FmcFlr.VortexCalibrActive AND NOT MAU_DumCon.DataOut.FillerFirstHalfPosReq
	AND NOT MAU_DumCon.DataOut.FillerSecondHalfPosReq AND NOT MAU_DumCon.DataOut.FillerReversePosReq THEN//V4.A.A.1.7.0//v999
	VAR_MNM_AutoStep := MNM_AutoWaitStart;
ELSIF NOT VAR_MNM_MachineStop OR VAR_MNM_AutoStopRequest THEN
	VAR_MNM_AutoStep := MNM_AutoMachineStopping;
ELSIF NOT MC_InputOutput.Network.Machine.Status.MachineRunning AND EDGEPOS(VAR_AutoStepCheck) THEN
	VAR_MNM_AutoStep := MNM_AutoCheckFillerInletHorn;
END_IF

TMR_TON_StartingHornElapsed.IN	:= FALSE;
MC_InputOutput.Network.Machine.Commands.MachineStart				:= FALSE;
MC_InputOutput.Network.Machine.Commands.StepByStepModalityRequest	:= FALSE;
MC_InputOutput.Network.Machine.Commands.PositioningModalityRequest	:= FALSE;
MC_InputOutput.Network.Machine.Commands.StepByStepSingleAxisModReq	:= FALSE;// V999 test
MC_InputOutput.Network.Machine.Commands.StepByStepSingleAxisRevModReq	:= FALSE;

VAR_MNM_HornFlrRequest	:= FALSE;
MNM.DataOut.StartLightFixRequest	:= FALSE;
MNM.DataOut.StartLightBlinkRequest	:= FALSE;
MNM.DataOut.FillingValvePositioningDone	:= FALSE;
MNM.DataOut.ReversePositioningDone	:= FALSE;//V4.A.A.1.7.0 -> taked from RMA
MNM.DataOut.DmcPositioningDone	:= FALSE;
//DOS.DataOut.AxisDisableRequest
//DOS.DataOut.AxisEnableRequest

//DOS.DataOut.PhasingWithoutDos;
//IF VAR_MNM_FillerPhasingHemaReq AND NOT (MC_InputOutput.Network.Machine.Status.MachineRunning) AND VAR_MNM_CocleaPhasingHemaDone THEN
//	VAR_MNM_CocleaPhasingPerValue := 74.0;
//ELSIF VAR_MNM_FillerPhasingHemaReq AND NOT (MC_InputOutput.Network.Machine.Status.MachineRunning) AND VAR_MNM_CocleaPhasingByPassDone THEN
//	VAR_MNM_CocleaPhasingPerValue := 0.0;
//ELSIF VAR_MNM_FillerPhasingHemaReq AND NOT (MC_InputOutput.Network.Machine.Status.MachineRunning) AND VAR_MNM_RinserPhasingHemaDone THEN
//	VAR_MNM_RinserPhasingPerValue := 74.0;
//ELSIF VAR_MNM_FillerPhasingHemaReq AND NOT (MC_InputOutput.Network.Machine.Status.MachineRunning) AND VAR_MNM_RinserPhasingByPassDone THEN
//	VAR_MNM_RinserPhasingPerValue := 0.0;
//END_IF

VAR_MNM_PccTestFirstHalf	:= 77;//set correct value of position, first position
VAR_MNM_PccTestSecondHalf	:= 27;//set correct value of position, second position
HMI_MNM_NumOfDmcInTangentSector1 := INT_TO_USINT(VAR_MNM_PccTestFirstHalf);
HMI_MNM_NumOfDmcInTangentSector2 := INT_TO_USINT(VAR_MNM_PccTestSecondHalf);
VAR_MNM_PccTestReversePos	:= 10;

CASE VAR_MNM_AutoStep OF
	MNM_AutoWaitStart:
		IF (VAR_MNM_MachineStart OR VAR_MNM_AutoStartRequest) AND VAR_MNM_MachineStop AND MC_InputOutput.Network.Machine.Status.EnableStart THEN
			VAR_MNM_AutoStep := MNM_AutoHornBlow;
		END_IF
		MNM.DataOut.StartLightBlinkRequest	:= NOT FmcFlr.FillingManualTestActive;

		IF IO_PB_FmcStep.ON AND FmcFlr.FillingManualTestActive THEN
			HMI_MNM_AxisStepByStepOffset	:= 1;
			VAR_MNM_AutoStep := MNM_AutoStepHornBlow;
		ELSIF VAR_MNM_AutoVortexCalibActive THEN
			VAR_MNM_AutoStep := MNM_AutoVortexCalibIdle;
		ELSIF FmcFlr.VortexCalibrActive THEN
			VAR_MNM_AutoStep := MNM_AutoVortexCalibHornBlow;
		ELSIF HMI_MNM_PB[PB_MNM_AxisStepByStep].ON THEN
			VAR_MNM_AutoStep := MNM_AutoStepHornBlow;
		ELSIF SFT.DataOut.FillingValvePositionReq THEN
			VAR_MNM_AutoStep := MNM_AutoFillingValvePosHornBlow;
		ELSIF MAU_DumCon.DataOut.FillerFirstHalfPosReq THEN//v999
			VAR_MNM_AutoStep := MNM_AutoFillerHalfPosConfig;//v999
		ELSIF MAU_DumCon.DataOut.FillerSecondHalfPosReq THEN
			VAR_MNM_AutoStep := MNM_AutoFillSecondHalfPosConfig;
		ELSIF MAU_DumCon.DataOut.FillerReversePosReq THEN
			VAR_MNM_AutoStep := MNM_AutoFillerReversePosConfig;
		END_IF

	MNM_AutoHornBlow:
		MNM.DataOut.StartLightFixRequest	:= TRUE;
		TMR_TON_StartingHornElapsed.IN		:= TRUE;
		VAR_MNM_HornFlrRequest	:= TRUE;

		IF NOT ((VAR_MNM_MachineStart OR VAR_MNM_AutoStartRequest) AND VAR_MNM_MachineStop AND MC_InputOutput.Network.Machine.Status.EnableStart) THEN
			VAR_MNM_AutoStep := MNM_AutoWaitStart;
		END_IF

		IF TMR_TON_StartingHornElapsed.Q THEN
			VAR_MNM_AutoStep := MNM_AutoMachineStart;
		END_IF

	MNM_AutoMachineStart:
		MC_InputOutput.Network.Machine.Commands.MachineStart := TRUE;
		MNM.DataOut.StartLightFixRequest	:= TRUE;

		IF MC_InputOutput.Network.Machine.Status.MachineRunning AND MC_InputOutput.Network.Machine.Status.MachineSynchro THEN
			VAR_MNM_AutoStep := MNM_AutoMachineRunningEmpty;
		END_IF

	MNM_AutoMachineRunningEmpty:	//Wait stop PB or Fault
		MC_InputOutput.Network.Machine.Commands.MachineStart := TRUE;
		MNM.DataOut.StartLightFixRequest	:= TRUE;

		IF MC_InputOutput.Network.Machine.Status.MachineRunning AND NOT SFT.DataOut.MachineEmpty THEN
			VAR_MNM_AutoStep	:= MNM_AutoMachineRunningFull;
		END_IF

		IF FmcFlr.VortexCalibrActive THEN
			VAR_MNM_AutoStep := MNM_AutoMachineStopping;
		END_IF

//		IF (DOS.DataOut.PhasingWithDos OR DOS.DataOut.PhasingWithoutDos) AND MC_InputOutput.Network.Machine.Status.MachineRunning THEN // Phasing req
//			VAR_MNM_AutoStep := MNM_AutoMachineColceaPashing; //first motor phased coclea
//		END_IF

		IF EDGEPOS(HMI_MNM_PB[PB_MNM_AxisInMotionAdjustment].ON) THEN
			MC_InputOutput.Network.Machine.Parameters.InMotionTimerValue	:= VAR_MNM_PAMValueTest;
			MC_InputOutput.Network.Machine.Commands.InMotionTimerModReq		:= TRUE;
			ALR[686].Active	:= TRUE;
		ELSIF MC_InputOutput.Network.Machine.Commands.InMotionTimerModReq AND MC_InputOutput.Network.Machine.Status.InMotionTimerDone THEN
			MC_InputOutput.Network.Machine.Commands.InMotionTimerModReq		:= FALSE;
			HMI_MNM_AxisInMotionAdjustment	:= 0.0;
			ALR[686].Active	:= FALSE;
		ELSIF NOT MC_InputOutput.Network.Machine.Commands.InMotionTimerModReq THEN
			ALR[686].Active	:= FALSE;
		END_IF

	MNM_AutoMachineColceaPashing:

		MC_InputOutput.Network.Machine.Commands.MachineStart := TRUE;
		MNM.DataOut.StartLightFixRequest	:= TRUE;

		HMI_MNM_AxisSelected		:= 113;//colea motor index for MC

		IF MC_InputOutput.Network.Machine.Status.EnableInMotionTimer AND DOS.DataOut.PhasingWithDos AND VAR_MNM_CocleaPhasingPerValue = 0.0 THEN
			VAR_MNM_CocleaPhasingHemaDone := FALSE;
			MC_InputOutput.Network.Machine.Parameters.InMotionTimerValue	:= VAR_MNM_PAMValueTest;
			MC_InputOutput.Network.Machine.Commands.InMotionTimerModReq		:= TRUE;
			ALR[686].Active	:= TRUE;//cambiare numero allarme
		ELSIF MC_InputOutput.Network.Machine.Status.EnableInMotionTimer AND DOS.DataOut.PhasingWithDos AND VAR_MNM_CocleaPhasingPerValue = 74.0 THEN
			ALR[686].Active	:= TRUE;
			VAR_MNM_AutoStep := MNM_AutoMachineRinserPashing;
		ELSIF	MC_InputOutput.Network.Machine.Status.EnableInMotionTimer AND DOS.DataOut.PhasingWithoutDos AND VAR_MNM_CocleaPhasingPerValue = 74.0 THEN
			MC_InputOutput.Network.Machine.Parameters.InMotionTimerValue	:= (LREAL_TO_REAL(CFG_MC.Mechanical.MachineStep) - VAR_MNM_PAMValueTest);
			MC_InputOutput.Network.Machine.Commands.InMotionTimerModReq		:= TRUE;
			ALR[686].Active	:= TRUE;
		ELSIF	MC_InputOutput.Network.Machine.Status.EnableInMotionTimer AND DOS.DataOut.PhasingWithoutDos AND VAR_MNM_CocleaPhasingPerValue = 0.0 THEN
			VAR_MNM_AutoStep := MNM_AutoMachineRinserPashing;
			ALR[686].Active	:= TRUE;
		ELSIF MC_InputOutput.Network.Machine.Commands.InMotionTimerModReq AND MC_InputOutput.Network.Machine.Status.InMotionTimerDone AND DOS.DataOut.PhasingWithDos THEN
			MC_InputOutput.Network.Machine.Commands.InMotionTimerModReq		:= FALSE;
			VAR_MNM_CocleaPhasingHemaDone := TRUE;
			VAR_MNM_AutoStep := MNM_AutoMachineRinserPashing;
		ELSIF MC_InputOutput.Network.Machine.Commands.InMotionTimerModReq AND MC_InputOutput.Network.Machine.Status.InMotionTimerDone AND DOS.DataOut.PhasingWithoutDos THEN
			MC_InputOutput.Network.Machine.Commands.InMotionTimerModReq		:= FALSE;
			VAR_MNM_CocleaPhasingPerValue := 0.0;
			VAR_MNM_AutoStep := MNM_AutoMachineRinserPashing;
		END_IF

//	MNM_AutoMachineStarWheel1Pashing: non serve per test
//
//		MC_InputOutput.Network.Machine.Commands.MachineStart := TRUE;
//		MNM.DataOut.StartLightFixRequest	:= TRUE;
//
//		IF MC_InputOutput.Network.Machine.Status.EnableInMotionTimer THEN
//			MC_InputOutput.Network.Machine.Parameters.InMotionTimerValue	:= VAR_MNM_PAMValueTest;
//			MC_InputOutput.Network.Machine.Commands.InMotionTimerModReq		:= TRUE;
//			MC_InputOutput.Network.Machine.Parameters.AxisSelectedOnHmi		:=
//			ALR[686].Active	:= TRUE;
//		ELSIF MC_InputOutput.Network.Machine.Commands.InMotionTimerModReq AND MC_InputOutput.Network.Machine.Status.InMotionTimerDone THEN
//			MC_InputOutput.Network.Machine.Commands.InMotionTimerModReq		:= FALSE;
//			VAR_MNM_AutoStep := MNM_AutoMachineRunningEmpty;
//			ALR[686].Active	:= FALSE;
//		END_IF

	MNM_AutoMachineRinserPashing:

		MC_InputOutput.Network.Machine.Commands.MachineStart := TRUE;
		MNM.DataOut.StartLightFixRequest	:= TRUE;

		HMI_MNM_AxisSelected		:= 114;//rinser motor index for MC

		IF MC_InputOutput.Network.Machine.Status.EnableInMotionTimer AND DOS.DataOut.PhasingWithDos AND VAR_MNM_RinserPhasingPerValue = 0 THEN
			MC_InputOutput.Network.Machine.Parameters.InMotionTimerValue	:= VAR_MNM_PAMValueTest;
			MC_InputOutput.Network.Machine.Commands.InMotionTimerModReq		:= TRUE;
			ALR[686].Active	:= TRUE;
		ELSIF MC_InputOutput.Network.Machine.Status.EnableInMotionTimer AND DOS.DataOut.PhasingWithDos AND VAR_MNM_RinserPhasingPerValue = 74.0 THEN
			ALR[686].Active	:= TRUE;
			VAR_MNM_AutoStep := MNM_AutoMachineRunningEmpty;
		ELSIF	MC_InputOutput.Network.Machine.Status.EnableInMotionTimer AND DOS.DataOut.PhasingWithoutDos AND VAR_MNM_RinserPhasingPerValue = 74.0 THEN
			MC_InputOutput.Network.Machine.Parameters.InMotionTimerValue	:= (LREAL_TO_REAL( CFG_MC.Mechanical.MachineStep) - VAR_MNM_PAMValueTest);
			MC_InputOutput.Network.Machine.Commands.InMotionTimerModReq		:= TRUE;
			ALR[686].Active	:= TRUE;
		ELSIF	MC_InputOutput.Network.Machine.Status.EnableInMotionTimer AND DOS.DataOut.PhasingWithoutDos AND VAR_MNM_RinserPhasingPerValue = 0.0 THEN
			VAR_MNM_AutoStep := MNM_AutoMachineRunningEmpty;
			ALR[686].Active	:= TRUE;
		ELSIF MC_InputOutput.Network.Machine.Commands.InMotionTimerModReq AND MC_InputOutput.Network.Machine.Status.InMotionTimerDone AND DOS.DataOut.PhasingWithDos THEN
			MC_InputOutput.Network.Machine.Commands.InMotionTimerModReq		:= FALSE;
			VAR_MNM_RinserPhasingPerValue := 74.0;
			VAR_MNM_AutoStep := MNM_AutoMachineRunningEmpty;
		ELSIF MC_InputOutput.Network.Machine.Commands.InMotionTimerModReq AND MC_InputOutput.Network.Machine.Status.InMotionTimerDone AND DOS.DataOut.PhasingWithoutDos  THEN
			MC_InputOutput.Network.Machine.Commands.InMotionTimerModReq		:= FALSE;
			VAR_MNM_RinserPhasingPerValue := 0.0;
			VAR_MNM_AutoStep := MNM_AutoMachineRunningEmpty;
		END_IF

	MNM_AutoMachineStarWheel2Phasing:

		MC_InputOutput.Network.Machine.Commands.MachineStart := TRUE;
		MNM.DataOut.StartLightFixRequest	:= TRUE;

		IF MC_InputOutput.Network.Machine.Status.EnableInMotionTimer THEN
			MC_InputOutput.Network.Machine.Parameters.InMotionTimerValue	:= VAR_MNM_PAMValueTest;
			MC_InputOutput.Network.Machine.Commands.InMotionTimerModReq		:= TRUE;
			MC_InputOutput.Network.Machine.Parameters.AxisSelectedOnHmi		:=
			ALR[686].Active	:= TRUE;
		ELSIF MC_InputOutput.Network.Machine.Commands.InMotionTimerModReq AND MC_InputOutput.Network.Machine.Status.InMotionTimerDone THEN
			MC_InputOutput.Network.Machine.Commands.InMotionTimerModReq		:= FALSE;
			HMI_MNM_AxisInMotionAdjustment	:= 0.0;
			ALR[686].Active	:= FALSE;
		END_IF

	MNM_AutoMachineRunningFull:	//Wait stop PB or Fault
		MC_InputOutput.Network.Machine.Commands.MachineStart := TRUE;
		MNM.DataOut.StartLightFixRequest	:= TRUE;

		IF MC_InputOutput.Network.Machine.Status.MachineRunning AND SFT.DataOut.MachineEmpty THEN
			VAR_MNM_AutoStep	:= MNM_AutoMachineRunningEmpty;
		END_IF

	MNM_AutoMachineStopping:
		IF NOT MC_InputOutput.Network.Machine.Status.MachineRunning THEN
			VAR_MNM_AutoStep := MNM_AutoWaitStart;
		END_IF

	MNM_AutoVortexCalibHornBlow:
		TMR_TON_StartingHornElapsed.IN	:= TRUE;
		VAR_MNM_HornFlrRequest	:= TRUE;

		IF TMR_TON_StartingHornElapsed.Q THEN
			VAR_MNM_AutoStep := MNM_AutoVortexCalibPosStart;
		END_IF

	MNM_AutoVortexCalibPosStart:
		MC_InputOutput.Network.Machine.Parameters.StepNumber	:= 1;
		MC_InputOutput.Network.Machine.Commands.StepByStepModalityRequest	:= TRUE;

		IF MC_InputOutput.Network.Machine.Status.StepByStepModalityActive THEN
			VAR_MNM_AutoStep := MNM_AutoVortexCalibPosWaitStop;
		END_IF

	MNM_AutoVortexCalibPosWaitStop:
		IF NOT MC_InputOutput.Network.Machine.Status.StepByStepModalityActive AND NOT MC_InputOutput.Network.Machine.Status.MachineRunning THEN
			VAR_MNM_AutoVortexCalibActive := TRUE;
			VAR_MNM_AutoStep := MNM_AutoVortexCalibIdle;
		END_IF

	MNM_AutoVortexCalibIdle:
		IF EDGEPOS(FmcFlr.FillerOneStepReq) THEN
			VAR_MNM_AutoStep := MNM_AutoStepFmcHornBlow;
		END_IF

		IF NOT FmcFlr.VortexCalibrActive THEN
			VAR_MNM_AutoVortexCalibActive := FALSE;
			VAR_MNM_AutoStep := MNM_AutoWaitStart;
		END_IF

	MNM_AutoStepFmcHornBlow:
		TMR_TON_StartingHornElapsed.IN	:= TRUE;
		VAR_MNM_HornFlrRequest	:= TRUE;

		IF TMR_TON_StartingHornElapsed.Q THEN
			FlrFmc.FillerOneStepReceived	:= FmcFlr.FillerOneStepReq;
			VAR_MNM_AutoStep := MNM_AutoStepFmcStart;
		END_IF

	MNM_AutoStepFmcStart:
		MC_InputOutput.Network.Machine.Parameters.StepNumber	:= 1;
		MC_InputOutput.Network.Machine.Commands.StepByStepModalityRequest	:= TRUE;

		IF MC_InputOutput.Network.Machine.Status.StepByStepModalityActive THEN
			VAR_MNM_AutoStep := MNM_AutoStepFmcWaitStop;
		END_IF

	MNM_AutoStepFmcWaitStop:
		IF NOT MC_InputOutput.Network.Machine.Status.StepByStepModalityActive AND NOT MC_InputOutput.Network.Machine.Status.MachineRunning THEN
			VAR_MNM_AutoStep := MNM_AutoVortexCalibIdle;
		END_IF

	MNM_AutoStepHornBlow:
		TMR_TON_StartingHornElapsed.IN	:= TRUE;
		VAR_MNM_HornFlrRequest	:= TRUE;

		IF TMR_TON_StartingHornElapsed.Q THEN
			VAR_MNM_AutoStep := MNM_AutoStepStart;
		END_IF

	MNM_AutoStepStart:
		MC_InputOutput.Network.Machine.Parameters.StepNumber	:= HMI_MNM_AxisStepByStepOffset;
		MC_InputOutput.Network.Machine.Commands.StepByStepModalityRequest	:= TRUE;

		IF MC_InputOutput.Network.Machine.Status.StepByStepModalityActive THEN
			VAR_MNM_AutoStep := MNM_AutoStepWaitStop;
		END_IF

	MNM_AutoStepWaitStop:
		IF NOT MC_InputOutput.Network.Machine.Status.StepByStepModalityActive AND NOT MC_InputOutput.Network.Machine.Status.MachineRunning THEN
			VAR_MNM_AutoStep := MNM_AutoWaitStart;
		END_IF

	MNM_AutoFillingValvePosHornBlow:
		TMR_TON_StartingHornElapsed.IN	:= TRUE;
		VAR_MNM_HornFlrRequest	:= TRUE;

		IF TMR_TON_StartingHornElapsed.Q THEN
			VAR_MNM_AutoStep := MNM_AutoFillingValvePosStart;
		END_IF

	MNM_AutoFillingValvePosStart:

		IF (HMI_PAC_1._132 + (HMI_PAC_1._100 - ((LREAL_TO_INT(MC_InputOutput.Network.Filler.Status.FillerAbsolutePosition / 360.0)) - SFT.DataOut.FillingValvePosValue)) > HMI_PAC_1._100) THEN
			MC_InputOutput.Network.Machine.Parameters.StepNumber := HMI_PAC_1._132 + (HMI_PAC_1._100 - ((LREAL_TO_INT(MC_InputOutput.Network.Filler.Status.FillerAbsolutePosition / 360.0)) - SFT.DataOut.FillingValvePosValue)) - HMI_PAC_1._100;
		ELSE
			MC_InputOutput.Network.Machine.Parameters.StepNumber := HMI_PAC_1._132 + (HMI_PAC_1._100 - ((LREAL_TO_INT(MC_InputOutput.Network.Filler.Status.FillerAbsolutePosition / 360.0)) - SFT.DataOut.FillingValvePosValue));
		END_IF
		IF MC_InputOutput.Network.Machine.Parameters.StepNumber > 0 THEN
			MC_InputOutput.Network.Machine.Commands.StepByStepModalityRequest	:= TRUE;
		ELSE
			VAR_MNM_AutoStep := MNM_AutoFillingValvePosWaitStop;
		END_IF

		IF MC_InputOutput.Network.Machine.Status.StepByStepModalityActive THEN
			VAR_MNM_AutoStep := MNM_AutoFillingValvePosWaitStop;
		END_IF

	MNM_AutoFillingValvePosWaitStop:

		MC_InputOutput.Network.Machine.Commands.StepByStepModalityRequest	:= FALSE;

		IF NOT MC_InputOutput.Network.Machine.Status.StepByStepModalityActive AND NOT MC_InputOutput.Network.Machine.Status.MachineRunning THEN
			MNM.DataOut.FillingValvePositioningDone	:= TRUE;
			VAR_MNM_AutoStep := MNM_AutoWaitStart;
		END_IF

	MNM_AutoFault:
		IF NOT (VAR_MNM_NormalStop OR VAR_MNM_QuickStop OR VAR_MNM_NormalStopWithJog OR VAR_MNM_QuickStopWithJog OR VAR_MNM_StopAfterEmpty OR VAR_MNM_StopIfNotEmpty) THEN
			VAR_MNM_AutoStep := MNM_AutoWaitStart;
		END_IF

	MNM_AutoCheckFillerInletHorn:
		TMR_TON_StartingHornElapsed.IN	:= TRUE;
		VAR_MNM_HornFlrRequest	:= TRUE;

		IF TMR_TON_StartingHornElapsed.Q THEN
			VAR_MNM_AutoStep := MNM_AutoCheckFillerInletStart;
		END_IF

	MNM_AutoCheckFillerInletStart:
		MC_InputOutput.Network.Machine.Parameters.StepNumber	:= HMI_PAC_1._001;
		MC_InputOutput.Network.Machine.Commands.StepByStepModalityRequest	:= TRUE;

		IF MC_InputOutput.Network.Machine.Status.StepByStepModalityActive THEN
			VAR_MNM_AutoStep := MNM_AutoCheckFillerInletStop;
		END_IF

	MNM_AutoCheckFillerInletStop:
		IF NOT MC_InputOutput.Network.Machine.Status.StepByStepModalityActive AND NOT MC_InputOutput.Network.Machine.Status.MachineRunning AND
			VAR_AutoStepCheckNext THEN
			VAR_MNM_AutoStep := MNM_AutoCheckFillerTangencyHorn;
		END_IF

	MNM_AutoCheckFillerTangencyHorn:
		TMR_TON_StartingHornElapsed.IN	:= TRUE;
		VAR_MNM_HornFlrRequest	:= TRUE;

		IF TMR_TON_StartingHornElapsed.Q THEN
			VAR_MNM_AutoStep := MNM_AutoCheckFillerTangencyStart;
		END_IF

	MNM_AutoCheckFillerTangencyStart:
		MC_InputOutput.Network.Machine.Parameters.StepNumber	:= (HMI_PAC_1._150 - SFT.DataOut.RinserBypassedPointer) - HMI_PAC_1._001;//V4.A.A.1.7.0
		MC_InputOutput.Network.Machine.Commands.StepByStepModalityRequest	:= TRUE;

		IF MC_InputOutput.Network.Machine.Status.StepByStepModalityActive THEN
			VAR_MNM_AutoStep := MNM_AutoCheckFillerTangencyStop;
		END_IF

	MNM_AutoCheckFillerTangencyStop:
		IF NOT MC_InputOutput.Network.Machine.Status.StepByStepModalityActive AND NOT MC_InputOutput.Network.Machine.Status.MachineRunning AND
			VAR_AutoStepCheckNext THEN
			VAR_MNM_AutoStep := MNM_AutoCheckFillerOutletHorn;
		END_IF

	MNM_AutoCheckFillerOutletHorn:
		TMR_TON_StartingHornElapsed.IN	:= TRUE;
		VAR_MNM_HornFlrRequest	:= TRUE;

		IF TMR_TON_StartingHornElapsed.Q THEN
			VAR_MNM_AutoStep := MNM_AutoCheckFillerOutletStart;
		END_IF

	MNM_AutoCheckFillerOutletStart:
		MC_InputOutput.Network.Machine.Parameters.StepNumber	:= HMI_PAC_1._006 - HMI_PAC_1._150;
		MC_InputOutput.Network.Machine.Commands.StepByStepModalityRequest	:= TRUE;

		IF MC_InputOutput.Network.Machine.Status.StepByStepModalityActive THEN
			VAR_MNM_AutoStep := MNM_AutoCheckFillerOutletStop;
		END_IF

	MNM_AutoCheckFillerOutletStop:
		IF NOT MC_InputOutput.Network.Machine.Status.StepByStepModalityActive AND NOT MC_InputOutput.Network.Machine.Status.MachineRunning AND
			VAR_AutoStepCheckNext THEN
			VAR_MNM_AutoStep := MNM_AutoCheckCapsReleaseHorn;
		END_IF

	MNM_AutoCheckCapsReleaseHorn:
		TMR_TON_StartingHornElapsed.IN	:= TRUE;
		VAR_MNM_HornFlrRequest	:= TRUE;

		IF TMR_TON_StartingHornElapsed.Q THEN
			VAR_MNM_AutoStep := MNM_AutoCheckCapsReleaseStart;
		END_IF

	MNM_AutoCheckCapsReleaseStart:
		MC_InputOutput.Network.Machine.Parameters.StepNumber	:= HMI_PAC_1._402 - HMI_PAC_1._006;
		MC_InputOutput.Network.Machine.Commands.StepByStepModalityRequest	:= TRUE;

		IF MC_InputOutput.Network.Machine.Status.StepByStepModalityActive THEN
			VAR_MNM_AutoStep := MNM_AutoCheckCapsReleaseStop;
		END_IF

	MNM_AutoCheckCapsReleaseStop:
		IF NOT MC_InputOutput.Network.Machine.Status.StepByStepModalityActive AND NOT MC_InputOutput.Network.Machine.Status.MachineRunning AND
			VAR_AutoStepCheckNext THEN
			VAR_MNM_AutoStep := MNM_AutoWaitStart;
		END_IF

	//Filler first hal configuration step v999
	MNM_AutoFillerHalfPosConfig://v999

		VAR_MNM_FlrFirstHalfRunning := TRUE;

		IF LREAL_TO_INT(MC_InputOutput.Network.Filler.Status.FillerAbsolutePosition / 360.0) < VAR_MNM_PccTestFirstHalf THEN //numero di valvola in tangenza quando valvola 1 è in posizione giusta per prima metà
			MC_InputOutput.Network.Machine.Parameters.StepNumber		:= VAR_MNM_PccTestFirstHalf - (LREAL_TO_INT(MC_InputOutput.Network.Filler.Status.FillerAbsolutePosition / 360.0));//Fra
		ELSE
			MC_InputOutput.Network.Machine.Parameters.StepNumber	:= (HMI_PAC_1._100 - (LREAL_TO_INT(MC_InputOutput.Network.Filler.Status.FillerAbsolutePosition / 360.0))) + VAR_MNM_PccTestFirstHalf;//Fra
		END_IF
		VAR_MNM_AutoStep := MNM_AutoFillerHalfPosHornBlow;

	MNM_AutoFillSecondHalfPosConfig://v999

		VAR_MNM_FlrSecondHalfRunning := TRUE;

		IF LREAL_TO_INT(MC_InputOutput.Network.Filler.Status.FillerAbsolutePosition / 360.0) < VAR_MNM_PccTestSecondHalf THEN //numero di valvola in tangenza quando valvola 1 è in posizione giusta per prima metà
			MC_InputOutput.Network.Machine.Parameters.StepNumber		:= VAR_MNM_PccTestSecondHalf - (LREAL_TO_INT(MC_InputOutput.Network.Filler.Status.FillerAbsolutePosition / 360.0));//Fra
		ELSE
			MC_InputOutput.Network.Machine.Parameters.StepNumber	:= (HMI_PAC_1._100 - (LREAL_TO_INT(MC_InputOutput.Network.Filler.Status.FillerAbsolutePosition / 360.0))) + VAR_MNM_PccTestSecondHalf;//Fra
		END_IF
		VAR_MNM_AutoStep := MNM_AutoFillerHalfPosHornBlow;

	MNM_AutoFillerHalfPosHornBlow://v999
		TMR_TON_StartingHornElapsed.IN	:= TRUE;
		VAR_MNM_HornFlrRequest	:= TRUE;

		IF TMR_TON_StartingHornElapsed.Q THEN
			VAR_MNM_AutoStep := MNM_AutoFillerHalfAxisStart;
		END_IF

	MNM_AutoFillerHalfAxisStart://v999
		MC_InputOutput.Network.Machine.Commands.StepByStepModalityRequest := TRUE;

		IF MC_InputOutput.Network.Machine.Status.StepByStepModalityActive THEN
			VAR_MNM_AutoStep := MNM_AutoFillerHalfWaitStop;
		END_IF
	MNM_AutoFillerHalfWaitStop://v999

		MC_InputOutput.Network.Machine.Commands.StepByStepModalityRequest:= FALSE;

		IF NOT MC_InputOutput.Network.Machine.Status.StepByStepModalityActive AND NOT MC_InputOutput.Network.Machine.Status.MachineRunning THEN
			MNM.DataOut.DmcPositioningDone	:= TRUE;
			IF NOT MAU_DumCon.DataOut.FillerSecondHalfPosReq AND NOT MAU_DumCon.DataOut.FillerFirstHalfPosReq THEN
				MNM.DataOut.DmcPositioningDone	:= FALSE;
				VAR_MNM_AutoStep := MNM_AutoWaitStart;
			END_IF
		END_IF

	MNM_AutoFillerReversePosConfig://v999

		VAR_MNM_FlrFirstHalfRunning := TRUE;

		HMI_MNM_AxisSelected := CFG_MC.Mechanical.ReferenceId.Filler + CST_FillerSubModuleHmiStart;

		MC_InputOutput.Network.Machine.Parameters.StepNumber		:= VAR_MNM_PccTestReversePos;//v999

		VAR_MNM_AutoStep := MNM_AutoFillerReversePosHornBlow;

	MNM_AutoFillSecondHalfRevPosConf:
		VAR_MNM_FlrSecondHalfRunning	:= TRUE;

		HMI_MNM_AxisSelected := CFG_MC.Mechanical.ReferenceId.Filler + CST_FillerSubModuleHmiStart;

		MC_InputOutput.Network.Machine.Parameters.StepNumber		:= VAR_MNM_PccTestReversePos;//v999

		VAR_MNM_AutoStep := MNM_AutoFillerReversePosHornBlow;

	MNM_AutoFillerReversePosHornBlow://v999
		TMR_TON_StartingHornElapsed.IN	:= TRUE;
		VAR_MNM_HornFlrRequest	:= TRUE;

		IF TMR_TON_StartingHornElapsed.Q THEN
			VAR_MNM_AutoStep := MNM_AutoFillerReverseAxisStart;
		END_IF

	MNM_AutoFillerReverseAxisStart://v999
		MC_InputOutput.Network.Machine.Commands.StepByStepSingleAxisRevModReq:= TRUE;

		IF MC_InputOutput.Network.Machine.Status.StepByStepSingleAxisRevModActive THEN
			VAR_MNM_AutoStep := MNM_AutoFillerReverseWaitStop;
		END_IF
	MNM_AutoFillerReverseWaitStop://v999

		MC_InputOutput.Network.Machine.Commands.StepByStepSingleAxisRevModReq:= FALSE;

		IF NOT MC_InputOutput.Network.Machine.Status.StepByStepSingleAxisRevModActive AND NOT MC_InputOutput.Network.Machine.Status.MachineRunning  THEN
			MNM.DataOut.ReversePositioningDone := TRUE;
			IF NOT MAU_DumCon.DataOut.FillerReversePosReq THEN
				MNM.DataOut.ReversePositioningDone	:= FALSE;
				VAR_MNM_AutoStep := MNM_AutoWaitStart;
			END_IF
		END_IF

END_CASE

TMR_TON_StartingHornElapsed(PT:= t#2s);

IF NOT FmcFlr.FillerOneStepReq THEN
	FlrFmc.FillerOneStepReceived	:= FALSE;
END_IF
END_STEP
ENTRY_ACTION
VAR_MNM_AutoStep := MNM_AutoWaitStart;
END_ACTION
TRANSITION IdleMode FROM MNMAuto TO MNMIdle:=
(NOT OPS.DataOut.FlrModeSelectorAuto AND NOT MC_InputOutput.Network.Machine.Status.MachineRunning) OR//V4 200.2.0
TMR_TON_TimeoutModality.Q
END_TRANSITION
(* @SFCISJUMP := 'MNMIdle' *)
STEP SpeedMng:
(*FIX SPEED FROM DMC*)
VAR_FixSpeed[1].Module			:= 2;
VAR_FixSpeed[1].Interruptible	:= FALSE;
VAR_FixSpeed[1].Value			:= HMI_PAM_1._003;
VAR_FixSpeed[1].Req				:= MAU_DumCon.DataOut.FixSpeedRequest;
VAR_FixSpeed[1].CmpMode			:= CST_LT;
(*FIX SPEED FROM PROCESS CPU*)
VAR_FixSpeed[2].Module			:= 2;
VAR_FixSpeed[2].Interruptible	:= TRUE;
VAR_FixSpeed[2].Value			:= SEL(CFG_Par.Process.BlendFill, SkdFlr.FixSpeedSP, CrbFlr.FixSpeedSP);
VAR_FixSpeed[2].Req				:= SEL(CFG_Par.Process.BlendFill, SkdFlr.FixSpeedRequest, CrbFlr.FixSpeedRequest);
VAR_FixSpeed[2].CmpMode			:= CST_EQ;
(*PROCESS REDUCE SPEED REQUEST*)
VAR_FixSpeed[3].Module			:= 0;
VAR_FixSpeed[3].Interruptible	:= NOT MNM.DataOut.ContBlockSpeedReached AND SFT.DataOut.ContBlockSpeedReq;
VAR_FixSpeed[3].Value			:= MAX(2000.0,(DINT_TO_REAL(HMI_MNM_FlrSpeedWidget.AutoSpeedReq) * HMI_PAM_1._000) / 100.0);
VAR_FixSpeed[3].Req				:= (ITC.DataOut.SlowDownReq OR SEL(CFG_Par.Process.BlendFill, SkdFlr.ReduceSpeedRequest, CrbFlr.ReduceSpeedRequest)) AND NOT SFT.DataOut.MachineEmpty;
VAR_FixSpeed[3].CmpMode			:= CST_EQ;
(*FIX SPEED FOR MCHINE EMPTY*)
VAR_FixSpeed[4].Module			:= 0;
VAR_FixSpeed[4].Interruptible	:= TRUE;
VAR_FixSpeed[4].Value			:= HMI_PAM_1._001;
VAR_FixSpeed[4].Req				:= SFT.DataOut.MachineEmpty AND HMI_CFG_PAM_1._001 AND NOT SkdFlr.FixSpeedRequest AND NOT MAU_DumCon.DataOut.FixSpeedRequest AND NOT CrbFlr.FixSpeedRequest;
VAR_FixSpeed[4].CmpMode			:= CST_EQ;
(*FIX SPEED FROM COP*)
VAR_FixSpeed[5].Module			:= 2;
VAR_FixSpeed[5].Interruptible	:= TRUE;
VAR_FixSpeed[5].Value			:= COP.DataOut.FixSpeedValue;
VAR_FixSpeed[5].Req				:= COP.DataOut.FixSpeedRequest AND NOT MAU_DumCon.DataOut.FixSpeedRequest;
VAR_FixSpeed[5].CmpMode			:= CST_EQ;
(*FIX SPEED FOR CAPPER EMPTYING*)
VAR_FixSpeed[6].Module			:= 2;
VAR_FixSpeed[6].Interruptible	:= FALSE;
VAR_FixSpeed[6].Value			:= HMI_PAM_1._007;
VAR_FixSpeed[6].Req				:= CAP.DataOut.SlowSpeedForEmptyReq AND NOT MAU_DumCon.DataOut.FixSpeedRequest;
VAR_FixSpeed[6].CmpMode			:= CST_EQ;
(*FIX SPEED FROM RINSER*)
VAR_FixSpeed[7].Module			:= 2;
VAR_FixSpeed[7].Interruptible	:= FALSE;
VAR_FixSpeed[7].Value			:= RNS.DataOut.FixSpeedValue;
VAR_FixSpeed[7].Req				:= RNS.DataOut.FixSpeedRequest;
VAR_FixSpeed[7].CmpMode			:= CST_EQ;
(*FIX SPEED FMC RECIPE DOWNLOAD REQ*)
VAR_FixSpeed[8].Module			:= 0;
VAR_FixSpeed[8].Interruptible	:= FALSE;
VAR_FixSpeed[8].Value			:= 74000.0;
VAR_FixSpeed[8].Req				:= (FmcFlr.FixSpeedRequestRecipeDownload OR FmcFlr.FixSpeedRequestChecking) AND NOT SFT.DataOut.MachineEmpty AND NOT MAU_DumCon.DataOut.FixSpeedRequest;
VAR_FixSpeed[8].CmpMode			:= CST_EQ;
(*FIX SPEED FROM CONTAINER BLOCK*)
VAR_FixSpeed[9].Module			:= 0;
VAR_FixSpeed[9].Interruptible	:= FALSE;
VAR_FixSpeed[9].Value			:= SFT.DataOut.ContBlockSpeedValue;
VAR_FixSpeed[9].Req				:= SFT.DataOut.ContBlockSpeedReq AND NOT MAU_DumCon.DataOut.FixSpeedRequest;
VAR_FixSpeed[9].CmpMode			:= CST_LE;
(*FIX SPEED FROM COP INLET*)
VAR_FixSpeed[10].Module			:= 2;
VAR_FixSpeed[10].Interruptible	:= FALSE;
VAR_FixSpeed[10].Value			:= SFT.DataOut.COPInletContBlockSpeedValue;
VAR_FixSpeed[10].Req			:= SFT.DataOut.COPInletContSlowSpeedReq AND NOT MAU_DumCon.DataOut.FixSpeedRequest;
VAR_FixSpeed[10].CmpMode		:= CST_EQ;
(*FIX SPEED FROM DOSER*) //v999hema
VAR_FixSpeed[11].Module			:= 2;
VAR_FixSpeed[11].Interruptible	:= FALSE;
VAR_FixSpeed[11].Value			:= DOS.DataOut.FixSpeedValue;
VAR_FixSpeed[11].Req			:= DOS.DataOut.FixSpeedRequest AND NOT MAU_DumCon.DataOut.FixSpeedRequest;
VAR_FixSpeed[11].CmpMode		:= CST_EQ;

MNM_MachineSpeedManagemant;

MNM.DataOut.DmcSpeedReqReached				:= VAR_FixSpeed[1].Reached;
MNM.DataOut.SkidSpeedReqReached				:= VAR_FixSpeed[2].Reached;
MNM.DataOut.SftSpeedReqReached				:= VAR_FixSpeed[3].Reached;
MNM.DataOut.EmptySpeedReached				:= VAR_FixSpeed[4].Reached;
MNM.DataOut.CopSpeedReqReached				:= VAR_FixSpeed[5].Reached OR (COP.DataOut.FixSpeedRequest AND MNM.DataOut.SkidSpeedReqReached) OR (VAR_FixSpeed[11].Reached AND DOS.DataOut.FixSpeedRequest);//v999hema
MNM.DataOut.CapSpeedReqReached				:= VAR_FixSpeed[6].Reached;
MNM.DataOut.RnsSpeedReqReached				:= VAR_FixSpeed[7].Reached;
MNM.DataOut.ContBlockSpeedReached			:= VAR_FixSpeed[9].Reached;
MNM.DataOut.COPInletContBlockSpeedReached	:= VAR_FixSpeed[10].Reached;

IF VAR_FixSpeedActive <> 0 THEN
	VAR_MNM_MachineSpeedRequest	:= VAR_ModuleSpeed.Machine;
ELSIF CvoFlr.OverSpeedFromInfeed (*AND CvoFlr.OverSpeedFromOutfeed*) THEN
	VAR_MNM_MachineSpeedRequest	:= VAR_ModuleSpeed.Machine;
ELSE
	IF CvoFlr.LineSpeedReference > 0 THEN
		VAR_MNM_MachineSpeedRequest	:= MIN(VAR_ModuleSpeed.Machine, INT_TO_REAL(CvoFlr.LineSpeedReference * 60));
	ELSE
		VAR_MNM_MachineSpeedRequest	:= VAR_ModuleSpeed.Machine;
	END_IF
END_IF
END_STEP
STEP MC_Interface:
MC_InputOutput.Network.Machine.Commands.HandShakeIn;

MC_InputOutput.Network.Machine.Commands.AlarmReset	:= AID.DataOut.Reset;

MC_InputOutput.Network.Machine.Commands.MachineQuickStop				:= (NOT VAR_MNM_QuickStop AND (NOT VAR_MNM_QuickStopWithJog OR OPS.DataOut.FlrModeSelectorJog));//v4 200.2.0

MC_InputOutput.Network.Filler.Commands.QuickStopFillerModule			:= NOT VAR_MNM_QuickStop AND (NOT VAR_MNM_QuickStopWithJog OR OPS.DataOut.FlrModeSelectorJog);

MC_InputOutput.Network.Machine.Commands.OnePitchShiftCommand;
MC_InputOutput.Network.Machine.Commands.KochModuleReady					:= IO_KochModuleOk.DI_Input;

MC_InputOutput.Network.Machine.Parameters.AutoAccelerationTime			:= HMI_PAM_1._011;
MC_InputOutput.Network.Machine.Parameters.AutoDecelerationTime			:= HMI_PAM_1._012;
MC_InputOutput.Network.Machine.Parameters.AutoSpeed						:= MAX(HMI_MNM_MinMachineSpeed, VAR_MNM_MachineSpeedRequest);
MC_InputOutput.Network.Machine.Parameters.JogSpeed						:= MAX(HMI_MNM_MinMachineJogSpeed, HMI_PAM_1._010);
MC_InputOutput.Network.Machine.Parameters.AxisSelectedOnHmi				:= HMI_MNM_AxisSelected;
MC_InputOutput.Network.Machine.Parameters.OffsetPositioning				:= HMI_MNM_AxisPositionOffset;

MC_InputOutput.Network.Filler.Parameters.AutoSpeedFillerModule			:= MAX(HMI_MNM_MinMachineSpeed, VAR_ModuleSpeed.Filler);
MC_InputOutput.Network.Filler.Parameters.FillerStepsNumber				:= HMI_PAC_1._100;
MC_InputOutput.Network.Filler.Parameters.RinserStepsNumber				:= HMI_PAC_1._200;
MC_InputOutput.Network.Filler.Parameters.DoserStepsNumber				;
MC_InputOutput.Network.Filler.Parameters.CapperStepsNumber				:= HMI_PAC_1._400;
MC_InputOutput.Network.Filler.Parameters.CrownerStepsNumber				:= HMI_PAC_1._300;

MC_InputOutput.Network.Filler.Parameters.FillerAbsolutePositionOffset	:= FmcFlr.OffsetSyncFVActTangInlet;
MC_InputOutput.Network.Filler.Parameters.RinserAbsolutePositionOffset	:= HMI_PAC_1._219;
IF CFG_Par.ClosingUnit.Capper.GreasingPumpPresent THEN//v4 200.2.0
	MC_InputOutput.Network.Filler.Parameters.CapperAbsolutePositionOffset	:= HMI_PAC_1._131;//v4 200.2.0
ELSE//v4 200.2.0
MC_InputOutput.Network.Filler.Parameters.CapperAbsolutePositionOffset	:= HMI_PAC_1._134;//v4 200.2.0
END_IF//v4 200.2.0
MC_InputOutput.Network.Filler.Parameters.DoserAbsolutePositionOffset	;
MC_InputOutput.Network.Filler.Parameters.CrownerAbsolutePositionOffset	:= HMI_PAC_1._133;

IF RNS.DataOut.ByPassRequest THEN//V4.A.A.1.7.0
	MC_InputOutput.Network.Filler.Commands.DisableRinserAxis := TRUE;//V4.A.A.1.7.0
ELSE//V4.A.A.1.7.0
	MC_InputOutput.Network.Filler.Commands.DisableRinserAxis := FALSE;//V4.A.A.1.7.0
END_IF//V4.A.A.1.7.0

//doser axis disable logic //v999hema
IF DOS.DataOut.AxisDisableRequest THEN //v999hema
	MC_InputOutput.Network.Filler.Commands.DisableDoserAxis := TRUE; //v999hema
ELSE //v999 test
	MC_InputOutput.Network.Filler.Commands.DisableDoserAxis := FALSE; //v999hema
END_IF //v999 test
//filler axis disable logic //v999hema
IF DOS.DataOut.FillerAxisDisableRequest THEN//biosgna ricordarsi che al cambio fra multi e auto modality bisogna riattivare l'asse filler. Se necessario successivamente riattivarlo //v999 test
	MC_InputOutput.Network.Filler.Commands.DisableFillerAxis := TRUE; //v999hema
ELSE //v999 test
	MC_InputOutput.Network.Filler.Commands.DisableFillerAxis := FALSE; //v999hema
END_IF //v999 test

IF TNK.DataOut.ProdMode OR COP.DataOut.RcpRunning OR SFT.DataOut.COPInletContConvEmptyRunning THEN
	MC_InputOutput.Network.Filler.Commands.VelocityAxisStop					:= FALSE;
	MC_InputOutput.Network.Outlet.Commands.VelocityAxisStop					:= FALSE;
ELSE
	MC_InputOutput.Network.Filler.Commands.VelocityAxisStop					:= TRUE;
	MC_InputOutput.Network.Outlet.Commands.VelocityAxisStop					:= TRUE;
END_IF

IF NOT FmcFlr.VortexCalibrActive THEN
	MC_InputOutput.Network.Machine.Parameters.StopPosition	:= MAX(0.1, HMI_PAM_1._013);
ELSE
	MC_InputOutput.Network.Machine.Parameters.StopPosition	:= MC_InputOutput.Network.Machine.Status.MachinePitch / 2.0;
END_IF

//CONTEINERS BLOCK
MC_InputOutput.Network.Machine.Parameters.Cam01OnValue			:= HMI_PAM_1._396;
HMI_PAM_1._397	:= INT_TO_REAL(FC_ReminderShift(REAL_TO_INT(HMI_PAM_1._396) + 180, 360, 0));
MC_InputOutput.Network.Machine.Parameters.Cam01OffValue			:= HMI_PAM_1._397;
MC_InputOutput.Network.Machine.Parameters.Cam01AdvTime			:= HMI_PAM_1._398;
MC_InputOutput.Network.Machine.Parameters.Cam01Pulse			:= REAL_TO_USINT(HMI_PAM_1._399);
HMI_MNM_CamName[1]							:= 1;
//CONTEINERS RELEASE//V4.A.A.1.7.0
MC_InputOutput.Network.Machine.Parameters.Cam02OnValue			:= HMI_PAM_1._400;
HMI_PAM_1._401	:= INT_TO_REAL(FC_ReminderShift(REAL_TO_INT(HMI_PAM_1._400) + 180, 360, 0));
MC_InputOutput.Network.Machine.Parameters.Cam02OffValue			:= HMI_PAM_1._401;
MC_InputOutput.Network.Machine.Parameters.Cam02AdvTime			:= HMI_PAM_1._402;
MC_InputOutput.Network.Machine.Parameters.Cam02Pulse			:= REAL_TO_USINT(HMI_PAM_1._403);
HMI_MNM_CamName[2]							:= 1;

//CAPS RELEASE / SECOND CROWN RELEASE(optional if it present)
MC_InputOutput.Network.Machine.Parameters.Cam03OnValue			:= HMI_PAM_1._404;
//HMI_PAM_1._405	:= INT_TO_REAL(FC_ReminderShift(REAL_TO_INT(HMI_PAM_1._404) + 180, 360, 0));
MC_InputOutput.Network.Machine.Parameters.Cam03OffValue			:= HMI_PAM_1._405;
MC_InputOutput.Network.Machine.Parameters.Cam03AdvTime			:= HMI_PAM_1._406;
MC_InputOutput.Network.Machine.Parameters.Cam03Pulse			:= REAL_TO_USINT(HMI_PAM_1._407);
HMI_MNM_CamName[3]							:= 1;

//CAPS CHECK
MC_InputOutput.Network.Machine.Parameters.Cam04OnValue			:= HMI_PAM_1._408;
//HMI_PAM_1._409	:= INT_TO_REAL(FC_ReminderShift(REAL_TO_INT(HMI_PAM_1._408) + 180, 360, 0));
MC_InputOutput.Network.Machine.Parameters.Cam04OffValue			:= HMI_PAM_1._409;
MC_InputOutput.Network.Machine.Parameters.Cam04AdvTime			:= HMI_PAM_1._410;
MC_InputOutput.Network.Machine.Parameters.Cam04Pulse			:= REAL_TO_USINT(HMI_PAM_1._411);
HMI_MNM_CamName[4]							:= 1;

//CONTAINERS EJECTION
MC_InputOutput.Network.Machine.Parameters.Cam05OnValue			:= HMI_PAM_1._412;
//HMI_PAM_1._413	:= INT_TO_REAL(FC_ReminderShift(REAL_TO_INT(HMI_PAM_1._412) + 180, 360, 0));to be defined
MC_InputOutput.Network.Machine.Parameters.Cam05OffValue			:= HMI_PAM_1._413;
MC_InputOutput.Network.Machine.Parameters.Cam05AdvTime			:= HMI_PAM_1._414;
MC_InputOutput.Network.Machine.Parameters.Cam05Pulse			:= REAL_TO_USINT(HMI_PAM_1._415);
IF CFG_Par.Rinser.NoBottleNoSpray THEN
	HMI_MNM_CamName[5]							:= 2;//v4 200.2.0
ELSE
	HMI_MNM_CamName[5]							:= 1;//v4 200.2.0
END_IF

//DATA MATRIX
MC_InputOutput.Network.Machine.Parameters.Cam06OnValue			:= HMI_PAM_1._416;
//HMI_PAM_1._417	:= INT_TO_REAL(FC_ReminderShift(REAL_TO_INT(HMI_PAM_1._416) + 180, 360, 0));
MC_InputOutput.Network.Machine.Parameters.Cam06OffValue			:= HMI_PAM_1._417;
MC_InputOutput.Network.Machine.Parameters.Cam06AdvTime			:= HMI_PAM_1._418;
MC_InputOutput.Network.Machine.Parameters.Cam06Pulse			:= REAL_TO_USINT(HMI_PAM_1._419);
HMI_MNM_CamName[6]							:= 1;

//CROWN RELEASE/ Second CAPS RELEASE(optional if it present)
MC_InputOutput.Network.Machine.Parameters.Cam07OnValue			:= HMI_PAM_1._420;
//HMI_PAM_1._421	:= INT_TO_REAL(FC_ReminderShift(REAL_TO_INT(HMI_PAM_1._420) + 180, 360, 0));//to be defined
MC_InputOutput.Network.Machine.Parameters.Cam07OffValue			:= HMI_PAM_1._421;
MC_InputOutput.Network.Machine.Parameters.Cam07AdvTime			:= HMI_PAM_1._422;
MC_InputOutput.Network.Machine.Parameters.Cam07Pulse			:= REAL_TO_USINT(HMI_PAM_1._423);
HMI_MNM_CamName[7]							:= 1;

//DUMMY CONTAINERS
MC_InputOutput.Network.Machine.Parameters.Cam08OnValue			:= HMI_PAM_1._424;
//HMI_PAM_1._425	:= INT_TO_REAL(FC_ReminderShift(REAL_TO_INT(HMI_PAM_1._424) + 180, 360, 0));//V4.A.A.1.7.0
MC_InputOutput.Network.Machine.Parameters.Cam08OffValue			:= HMI_PAM_1._425;
MC_InputOutput.Network.Machine.Parameters.Cam08AdvTime			:= HMI_PAM_1._426;
MC_InputOutput.Network.Machine.Parameters.Cam08Pulse			:= REAL_TO_USINT(HMI_PAM_1._427);
HMI_MNM_CamName[8]												:= 1;

// FCI - Clock//V4.A.A.1.7.0
MC_InputOutput.Network.Machine.Parameters.Cam09OnValue			:= HMI_PAM_1._428;
//HMI_PAM_1._429	:= INT_TO_REAL(FC_ReminderShift(REAL_TO_INT(HMI_PAM_1._428) + 180, 360, 0));to be defined
MC_InputOutput.Network.Machine.Parameters.Cam09OffValue			:= HMI_PAM_1._429;
MC_InputOutput.Network.Machine.Parameters.Cam09AdvTime			:= HMI_PAM_1._430;
MC_InputOutput.Network.Machine.Parameters.Cam09Pulse			:= REAL_TO_USINT(HMI_PAM_1._431);
HMI_MNM_CamName[9]							:= 1;

//FCI - Fine pulse
MC_InputOutput.Network.Machine.Parameters.Cam10OnValue			:= HMI_PAM_1._432;
//HMI_PAM_1._433	:= INT_TO_REAL(FC_ReminderShift(REAL_TO_INT(HMI_PAM_1._432) + 180, 360, 0));to be defined
MC_InputOutput.Network.Machine.Parameters.Cam10OffValue			:= HMI_PAM_1._433;
MC_InputOutput.Network.Machine.Parameters.Cam10AdvTime			:= HMI_PAM_1._434;
MC_InputOutput.Network.Machine.Parameters.Cam10Pulse			:= REAL_TO_USINT(HMI_PAM_1._435);
HMI_MNM_CamName[10]							:= 1;
//DOSER- camma doser v999hema
MC_InputOutput.Network.Machine.Parameters.Cam11OnValue			:= HMI_PAM_1._436;
//HMI_PAM_1._437	:= INT_TO_REAL(FC_ReminderShift(REAL_TO_INT(HMI_PAM_1._436) + 180, 360, 0));//V4.A.A.1.7.0 to be defined
MC_InputOutput.Network.Machine.Parameters.Cam11OffValue			:= HMI_PAM_1._437;
MC_InputOutput.Network.Machine.Parameters.Cam11AdvTime			:= HMI_PAM_1._438;
MC_InputOutput.Network.Machine.Parameters.Cam11Pulse			:= REAL_TO_USINT(HMI_PAM_1._439);
HMI_MNM_CamName[11]							:= 1;//V4.A.A.1.7.0
END_STEP
STEP Fan:
FillerFanMain(
IN_ConfigPresent	:= CFG_Par.Motors.CoolingFan.Filler.Main.Present,
IN_Enable			:= OPS.DataOut.FlrDoorsOk,
IN_AutoCnd			:= CFG_Par.Motors.CoolingFan.Filler.Main.CommandPresent,
IN_Reset			:= AID.DataOut.Reset,
IN_FBKDelay			:= t#500ms,
IO					:= IO_MNM_MotionFan.Filler.Main
);

FillerFanIn1(
IN_ConfigPresent	:= CFG_Par.Motors.CoolingFan.Filler.In[1].Present,
IN_Enable			:= OPS.DataOut.FlrDoorsOk,
IN_AutoCnd			:= CFG_Par.Motors.CoolingFan.Filler.In[1].CommandPresent,
IN_Reset			:= AID.DataOut.Reset,
IN_FBKDelay			:= t#500ms,
IO					:= IO_MNM_MotionFan.Filler.In1
);

FillerFanIn2(
IN_ConfigPresent	:= CFG_Par.Motors.CoolingFan.Filler.In[2].Present,
IN_Enable			:= OPS.DataOut.FlrDoorsOk,
IN_AutoCnd			:= CFG_Par.Motors.CoolingFan.Filler.In[2].CommandPresent,
IN_Reset			:= AID.DataOut.Reset,
IN_FBKDelay			:= t#500ms,
IO					:= IO_MNM_MotionFan.Filler.In2
);

FillerFanIn3(
IN_ConfigPresent	:= CFG_Par.Motors.CoolingFan.Filler.In[3].Present,
IN_Enable			:= OPS.DataOut.FlrDoorsOk,
IN_AutoCnd			:= CFG_Par.Motors.CoolingFan.Filler.In[3].CommandPresent,
IN_Reset			:= AID.DataOut.Reset,
IN_FBKDelay			:= t#500ms,
IO					:= IO_MNM_MotionFan.Filler.In3
);

FillerFanIn4(
IN_ConfigPresent	:= CFG_Par.Motors.CoolingFan.Filler.In[4].Present,
IN_Enable			:= OPS.DataOut.FlrDoorsOk,
IN_AutoCnd			:= CFG_Par.Motors.CoolingFan.Filler.In[4].CommandPresent,
IN_Reset			:= AID.DataOut.Reset,
IN_FBKDelay			:= t#500ms,
IO					:= IO_MNM_MotionFan.Filler.In4
);

FillerFanIn5(
IN_ConfigPresent	:= CFG_Par.Motors.CoolingFan.Filler.In[5].Present,
IN_Enable			:= OPS.DataOut.FlrDoorsOk,
IN_AutoCnd			:= CFG_Par.Motors.CoolingFan.Filler.In[5].CommandPresent,
IN_Reset			:= AID.DataOut.Reset,
IN_FBKDelay			:= t#500ms,
IO					:= IO_MNM_MotionFan.Filler.In5
);

FillerFanIn7(
IN_ConfigPresent	:= CFG_Par.Motors.CoolingFan.Filler.In[7].Present,
IN_Enable			:= OPS.DataOut.FlrDoorsOk,
IN_AutoCnd			:= CFG_Par.Motors.CoolingFan.Filler.In[7].CommandPresent,
IN_Reset			:= AID.DataOut.Reset,
IN_FBKDelay			:= t#500ms,
IO					:= IO_MNM_MotionFan.Filler.In7
);

FillerFanIn8(
IN_ConfigPresent	:= CFG_Par.Motors.CoolingFan.Filler.In[8].Present,
IN_Enable			:= OPS.DataOut.FlrDoorsOk,
IN_AutoCnd			:= CFG_Par.Motors.CoolingFan.Filler.In[8].CommandPresent,
IN_Reset			:= AID.DataOut.Reset,
IN_FBKDelay			:= t#500ms,
IO					:= IO_MNM_MotionFan.Filler.In8
);

FillerFanIn9(
IN_ConfigPresent	:= CFG_Par.Motors.CoolingFan.Filler.In[9].Present,
IN_Enable			:= OPS.DataOut.FlrDoorsOk,
IN_AutoCnd			:= CFG_Par.Motors.CoolingFan.Filler.In[9].CommandPresent,
IN_Reset			:= AID.DataOut.Reset,
IN_FBKDelay			:= t#500ms,
IO					:= IO_MNM_MotionFan.Filler.In9
);

FillerFanIn10(
IN_ConfigPresent	:= CFG_Par.Motors.CoolingFan.Filler.In[10].Present,
IN_Enable			:= OPS.DataOut.FlrDoorsOk,
IN_AutoCnd			:= CFG_Par.Motors.CoolingFan.Filler.In[10].CommandPresent,
IN_Reset			:= AID.DataOut.Reset,
IN_FBKDelay			:= t#500ms,
IO					:= IO_MNM_MotionFan.Filler.In10
);

FillerFanOut1(
IN_ConfigPresent	:= CFG_Par.Motors.CoolingFan.Filler.Out[1].Present,
IN_Enable			:= OPS.DataOut.FlrDoorsOk,
IN_AutoCnd			:= CFG_Par.Motors.CoolingFan.Filler.Out[1].CommandPresent,
IN_Reset			:= AID.DataOut.Reset,
IN_FBKDelay			:= t#500ms,
IO					:= IO_MNM_MotionFan.Filler.Out1
);

FillerFanOut2(
IN_ConfigPresent	:= CFG_Par.Motors.CoolingFan.Filler.Out[2].Present,
IN_Enable			:= OPS.DataOut.FlrDoorsOk,
IN_AutoCnd			:= CFG_Par.Motors.CoolingFan.Filler.Out[2].CommandPresent,
IN_Reset			:= AID.DataOut.Reset,
IN_FBKDelay			:= t#500ms,
IO					:= IO_MNM_MotionFan.Filler.Out2
);

FillerFanOut3(
IN_ConfigPresent	:= CFG_Par.Motors.CoolingFan.Filler.Out[3].Present,
IN_Enable			:= OPS.DataOut.FlrDoorsOk,
IN_AutoCnd			:= CFG_Par.Motors.CoolingFan.Filler.Out[3].CommandPresent,
IN_Reset			:= AID.DataOut.Reset,
IN_FBKDelay			:= t#500ms,
IO					:= IO_MNM_MotionFan.Filler.Out3
);

FillerFanOut4(
IN_ConfigPresent	:= CFG_Par.Motors.CoolingFan.Filler.Out[4].Present,
IN_Enable			:= OPS.DataOut.FlrDoorsOk,
IN_AutoCnd			:= CFG_Par.Motors.CoolingFan.Filler.Out[4].CommandPresent,
IN_Reset			:= AID.DataOut.Reset,
IN_FBKDelay			:= t#500ms,
IO					:= IO_MNM_MotionFan.Filler.Out4
);
END_STEP
STEP HmiData:

HMI_MNM_MachineSpeedAct	:= MC_InputOutput.Network.Machine.Status.ActualSpeed;//v4 200.2.0

HMI_MNM_FlrSpeedWidget.Visibility		:= NOT HMI_CmdBar_PB[PB_FillerLabellerCoupling].LampON AND NOT HMI_CmdBar_PB[PB_FillerBlowerCoupling].LampON;
IF MC_InputOutput.Network.Machine.Status.AutoModalityActive THEN
	HMI_MNM_FlrSpeedWidget.ActualSpeed		:= REAL_TO_DINT(MC_InputOutput.Network.Machine.Status.ActualSpeed);
ELSIF MC_InputOutput.Network.Machine.Status.MultiModalityActive THEN
	HMI_MNM_FlrSpeedWidget.ActualSpeed		:= REAL_TO_DINT(MC_InputOutput.Network.Filler.Status.Velocity);
ELSIF MC_InputOutput.Network.Machine.Status.JogModalityActive THEN
	HMI_MNM_FlrSpeedWidget.ActualSpeed		:= REAL_TO_DINT(MC_InputOutput.Network.Machine.Status.ActualSpeed);
END_IF

HMI_MNM_FlrSpeedWidget.Modality			:= OPS.DataOut.FlrModeSelectorJog;

IF EDGEPOS(OPS.DataOut.FlrModeSelectorJog) THEN
	HMI_MNM_FlrSpeedWidget.JogSpeedReq	:= REAL_TO_DINT(HMI_PAM_1._010);
	VAR_MNM_JogSpeedOld					:= HMI_PAM_1._010;
ELSIF OPS.DataOut.FlrModeSelectorJog THEN
	IF DINT_TO_REAL(HMI_MNM_FlrSpeedWidget.JogSpeedReq) <> VAR_MNM_JogSpeedOld THEN
		HMI_PAM_1._010 		:= DINT_TO_REAL(HMI_MNM_FlrSpeedWidget.JogSpeedReq);
		VAR_MNM_JogSpeedOld	:= HMI_PAM_1._010;
	ELSIF HMI_PAM_1._010 <> VAR_MNM_JogSpeedOld THEN
		HMI_MNM_FlrSpeedWidget.JogSpeedReq	:= REAL_TO_DINT(HMI_PAM_1._010);
		VAR_MNM_JogSpeedOld					:= HMI_PAM_1._010;
	END_IF
END_IF

(* Filler Status *)
IF OPS.DataOut.SelModeChange THEN
	HMI_MNM_FlrSpeedWidget.Status	:= 0;
ELSIF OPS.DataOut.FlrModeSelectorAuto THEN
	HMI_MNM_FlrSpeedWidget.Status	:= 1;
ELSIF OPS.DataOut.FlrModeSelectorJog THEN
	HMI_MNM_FlrSpeedWidget.Status	:= 2;
ELSIF OPS.DataOut.FlrModeSelectorAdjustment THEN
	HMI_MNM_FlrSpeedWidget.Status	:= 3;
END_IF

HMI_MNM_MachinePitch	:= MC_InputOutput.Network.Machine.Status.MachinePitch;
HMI_MNM_MaxMachineSpeed := MC_InputOutput.Network.Machine.Status.MachineMaxSpeed;
HMI_MNM_MachinePosition;	//COMPLETARE

HMI_MNM_PB[PB_MNM_AxisPositioning].Visibility	:= TRUE;
HMI_MNM_PB[PB_MNM_AxisPositioning].Enable		:= OPS.DataOut.FlrModeSelectorAdjustment AND OPS.DataOut.DoorsOk AND OPS.DataOut.EmergencyOk AND
													MC_InputOutput.Network.Machine.Status.EnablePositioning AND SFT.DataOut.MachineEmpty AND (HMI_MNM_AxisPositionOffset <> 0.0);
HMI_MNM_PB[PB_MNM_AxisPositioning].LampON		:= MC_InputOutput.Network.Machine.Status.PositioningModalityActive OR MC_InputOutput.Network.Machine.Commands.PositioningModalityRequest OR HMI_MNM_PB[PB_MNM_AxisPositioning].ON;

HMI_MNM_PB[PB_MNM_AxisHoming].Visibility	:= TRUE;
HMI_MNM_PB[PB_MNM_AxisHoming].Enable		:= OPS.DataOut.FlrModeSelectorAdjustment AND OPS.DataOut.DoorsOk AND OPS.DataOut.EmergencyOk AND
												MC_InputOutput.Network.Machine.Status.EnableHoming;
HMI_MNM_PB[PB_MNM_AxisHoming].LampON		:= MC_InputOutput.Network.Machine.Status.SelectiveHomeModalityActive OR MC_InputOutput.Network.Machine.Commands.SelectiveHomeModalityRequest OR HMI_MNM_PB[PB_MNM_AxisHoming].ON;

HMI_MNM_PB[PB_MNM_AxisStepByStep].Visibility	:= TRUE;
HMI_MNM_PB[PB_MNM_AxisStepByStep].Enable		:= MC_InputOutput.Network.Machine.Status.AutoModalityActive AND OPS.DataOut.DoorsOk AND OPS.DataOut.EmergencyOk AND
													NOT MC_InputOutput.Network.Machine.Status.MachineRunning AND MC_InputOutput.Network.Machine.Status.EnableStepByStep AND
													(HMI_MNM_AxisStepByStepOffset <> 0);
HMI_MNM_PB[PB_MNM_AxisStepByStep].LampON		:= (MC_InputOutput.Network.Machine.Status.StepByStepModalityActive OR MC_InputOutput.Network.Machine.Commands.StepByStepModalityRequest) AND
													((VAR_MNM_AutoStep = MNM_AutoStepHornBlow) OR (VAR_MNM_AutoStep = MNM_AutoStepStart) OR (VAR_MNM_AutoStep = MNM_AutoStepWaitStop));

//Footbar Filler
HMI_MNM_PB[PB_MNM_FootboardPosition].Visibility	:= CFG_Par.Motors.FootbarPresent;
HMI_MNM_PB[PB_MNM_FootboardPosition].Enable		:= OPS.DataOut.FlrModeSelectorAdjustment AND OPS.DataOut.DoorsOk AND OPS.DataOut.EmergencyOk AND SFT.DataOut.MachineEmpty AND
													NOT MC_InputOutput.Network.Machine.Status.MachineRunning AND MC_InputOutput.Network.Machine.Status.EnableStepByStep AND
													MC_InputOutput.Network.Filler.Status.FillerAbsolutePositionValid AND (LREAL_TO_INT(MC_InputOutput.Network.Filler.Status.FillerAbsolutePosition / 360.0) <> HMI_PAC_1._130);
HMI_MNM_PB[PB_MNM_FootboardPosition].LampON		:= (MC_InputOutput.Network.Machine.Status.StepByStepSingleAxisModeActive OR MC_InputOutput.Network.Machine.Commands.StepByStepSingleAxisModReq) AND
													VAR_MNM_AdjAxisFillerFootBar;//V4.A.A.1.7.0

HMI_MNM_PB[PB_MNM_AxisInMotionAdjustment].Visibility	:= FALSE;
HMI_MNM_PB[PB_MNM_AxisInMotionAdjustment].Enable		:= (MC_InputOutput.Network.Machine.Parameters.AxisSelectedOnHmi = 99) AND
															MC_InputOutput.Network.Machine.Status.AutoCombiModalityActive AND OPS.DataOut.FlrModeSelectorAuto AND OPS.DataOut.DoorsOk AND OPS.DataOut.EmergencyOk AND
															MC_InputOutput.Network.Machine.Status.MachineRunning AND MC_InputOutput.Network.Machine.Status.EnableInMotionTimer AND SFT.DataOut.CombiEmpty;
HMI_MNM_PB[PB_MNM_AxisInMotionAdjustment].LampON		:= MC_InputOutput.Network.Machine.Commands.InMotionTimerModReq;

IF SFT.DataOut.MachineEmpty THEN
	HMI_MNM_MinInMotionAdjustement	:= -40.0;
	HMI_MNM_MaxInMotionAdjustement	:= 40.0;
ELSE
	HMI_MNM_MinInMotionAdjustement	:= -10.0;
	HMI_MNM_MaxInMotionAdjustement	:= 10.0;
END_IF

HMI_MNM_PB[PB_MNM_BrakeRelease].Visibility	:= HMI_MC_GenericAxisData.xMotorWithBrake;
HMI_MNM_PB[PB_MNM_BrakeRelease].Enable		:= OPS.DataOut.FlrModeSelectorAdjustment AND MC_InputOutput.Network.Machine.Status.EnableBrakeRelease;
HMI_MNM_PB[PB_MNM_BrakeRelease].LampON		:= MC_InputOutput.Network.Machine.Commands.BrakeReleaseModalityRequest;

HMI_MNM_PB[PB_MNM_VelocityTest].Visibility	:= TRUE;
HMI_MNM_PB[PB_MNM_VelocityTest].Enable		:= (OPS.DataOut.FlrModeSelectorAdjustment AND MC_InputOutput.Network.Machine.Status.EnableVelocity) OR MC_InputOutput.Network.Machine.Commands.VelocityModalityRequest;
HMI_MNM_PB[PB_MNM_VelocityTest].LampON		:= MC_InputOutput.Network.Machine.Commands.VelocityModalityRequest;

HMI_MNM_PB[PB_MNM_RinserFootboardPosition].Visibility      := 	CFG_Par.Rinser.FootbarPresent;
HMI_MNM_PB[PB_MNM_RinserFootboardPosition].Enable          := 	OPS.DataOut.FlrModeSelectorAdjustment AND OPS.DataOut.DoorsOk AND OPS.DataOut.EmergencyOk AND
																NOT MC_InputOutput.Network.Machine.Status.MachineRunning AND MC_InputOutput.Network.Machine.Status.EnableStepByStep AND
                                                           	MC_InputOutput.Network.Filler.Status.RinserAbsolutePositionValid AND (LREAL_TO_INT(MC_InputOutput.Network.Filler.Status.RinserAbsolutePosition / 360.0) <> HMI_PAC_1._130);
HMI_MNM_PB[PB_MNM_RinserFootboardPosition].LampON          := 	(MC_InputOutput.Network.Machine.Status.StepByStepSingleAxisModeActive OR MC_InputOutput.Network.Machine.Commands.StepByStepSingleAxisModReq) AND
																VAR_MNM_AdjAxisRinserFootBar;
END_STEP
STEP InletConveyor:
END_STEP
TRANSITION PAO Conveyor VFD FROM InletConveyor TO InletConveyorVFD:=
CFG_Par.Motors.ConveyorVFD AND CFG_Par.Machine.Type.SRMA
END_TRANSITION
STEP InletConveyorVFD:
InletConveyorVar_VFD;
InletConveyorDigitalIn;
InletConveyorAlarm;

//IF VAR_MNM_ConveyorProduction THEN //v1.6//Master Bottle +PET
InletConveyorSeq_Run_VFD;
//ELSIF VAR_MNM_ConveyorClean THEN //v1.6//Master Bottle +PET
//	OutletConveyorSeq_Cleaning_VFD; //v1.6//Master Bottle +PET
//ELSE //v1.6//Master Bottle +PET
//	OutletConveyorSeq_Idle_VFD; //v1.6//Master Bottle +PET
//END_IF //v1.6//Master Bottle +PET

InletConveyorMotors_VFD;
InletConveyorDataOut_VFD;
InletConveyorAlarm_VFD;
InletConveyorHMI;
END_STEP
TRANSITION FROM InletConveyorVFD TO InletConveyor:=
FALSE
END_TRANSITION
(* @SFCISJUMP := 'InletConveyor' *)
STEP OutletConveyor:
END_STEP
TRANSITION PAO Conveyor VFD FROM OutletConveyor TO ConveyorVFD:=
CFG_Par.Motors.ConveyorVFD
END_TRANSITION
STEP ConveyorVFD:
OutletConveyorVar_VFD;
OutletConveyorDigitalIn;

//IF VAR_MNM_ConveyorProduction THEN //v1.6
	OutletConveyorSeq_Run_VFD;
//ELSIF VAR_MNM_ConveyorClean THEN //v1.6
//	OutletConveyorSeq_Cleaning_VFD; //v1.6
//ELSE //v1.6
//	OutletConveyorSeq_Idle_VFD; //v1.6
//END_IF //v1.6

OutletConveyorMotors_VFD;
OutletConveyorInterchange;
OutletConveyorDataOut_VFD;
OutletConveyorAlarm_VFD;
OutletConveyorHMI;
END_STEP
TRANSITION FROM ConveyorVFD TO OutletConveyor:=
FALSE
END_TRANSITION
(* @SFCISJUMP := 'OutletConveyor' *)
STEP DataTo:
MNM_DataOut;
MNM_MotionAlarm;
MNM_MotionModuleAlarm;
MNM_Alarm;
END_STEP
TRANSITION FROM (MNMVar,SpeedMng,MC_Interface,Fan,HmiData,DataTo) TO MNMInit:=
FALSE
END_TRANSITION
(* @SFCISJUMP := 'MNMInit' *)
END_PROGRAM
```

#### Variables.var - Local variables
```iecst
(*MAIN MOTORIZATION Variables*)
VAR
	VAR_MNM_MachineSpeedRequest : REAL;
	VAR_MNM_AdjustmentStep : MNM_AdjustmentStep; (*V4.A.A.1.7.0*)
	VAR_MNM_AutoStep : MNM_AutoStep;
	VAR_MNM_AutoCombiStep : MNM_AutoCombiStep;
	VAR_MNM_JogStep : MNM_JogStep;
	VAR_MNM_JogCombiStep : MNM_JogCombiStep;
	VAR_MNM_FlrMultiStep : MNM_MultiStep;
	VAR_MNM_FlrInletMultiStep : MNM_MultiStep;
	VAR_MNM_FlrSecondHalfRunning : BOOL;
	VAR_MNM_FlrRephasingPosition : USINT;
	VAR_MNM_FlrFirstHalfRunning : BOOL;
	VAR_MNM_FpMachineStartPb : BOOL;
	VAR_MNM_MachineStart : BOOL;
	VAR_MNM_MachineStopRequest : BOOL; (*V4.A.A.1.6.6*)
	VAR_MNM_MachineStop : BOOL;
END_VAR
(*FAULT VARIABLES*)
(*Machine*)
VAR
	VAR_MNM_NormalStop : BOOL;
	VAR_MNM_QuickStop : BOOL;
	VAR_MNM_NormalStopWithJog : BOOL;
	VAR_MNM_NormalWithJogMnt : BOOL; (*V4.A.A.1.6.13*)
	VAR_MNM_QuickStopWithJog : BOOL;
	VAR_MNM_StopIfNotEmpty : BOOL;
	VAR_MNM_StopAfterEmpty : BOOL;
	VAR_MNM_DisengageForStop : BOOL;
	VAR_MNM_HornFlrRequest : BOOL;
	VAR_MNM_PAMValueTest : REAL; (*variabile di test*)
	VAR_MNM_AutoStartRequest : BOOL;
	VAR_MNM_AutoStopRequest : BOOL;
	VAR_MNM_FlrAutoStartRequest : BOOL;
	VAR_MNM_FlrAutoStopRequest : BOOL;
	VAR_MNM_AutoVortexCalibActive : BOOL;
	TMR_TON_StartingHornElapsed : TON;
	VAR_MNM_AdjAxisRinserFootBar : BOOL; (*V4.A.A.1.7.0*)
	VAR_MNM_AdjAxisFillerFootBar : BOOL; (*V4.A.A.1.7.0*)
	VAR_MNM_AdjAxisPositionOffset : REAL;
	VAR_i : UINT;
	VAR_MNM_JogSpeedOld : REAL; (*V4.A.A.1.7.0*)
	TMR_TON_TimeoutModality : TON;
	VAR_MNM_CapperPosAux : BOOL; (*V4.A.A.1.6.12h*)
	VAR_MNM_CoupledDesychroReq : BOOL; (*V4.A.A.1.7.0*)
END_VAR
(*CONVEYOR Variables*)
VAR
	VAR_MNM_MachineSpeedRequest1 : REAL; (*Master nuovo*)
	VAR_MNM_InFixSpeedReq1 : BOOL; (*Master nuovo*)
	VAR_MNM_ConveyorProduction : BOOL;
	VAR_MNM_ConveyorClean : BOOL;
	FB_ScalConveyorInlet : LCRLimScal; (*Master nuovo*)
	FB_ScalConveyor : LCRLimScal;
	VAR_AutoStepCheckNext : BOOL;
	VAR_AutoStepCheck : BOOL;
	VAR_MNM_InletConveyorSeq_VFD : MNM_InletConveyorVFD; (*1.6*)
	VAR_MNM_OutletConveyorSeq_VFD : MNM_OutletConveyorVFD; (*1.6*)
	VAR_MNM_OptionNoGripper : BOOL; (*V1.61 - inserire CFG_Pao?*)
	VAR_MNM_InCvrAlarm : BOOL; (*1.6*) (*Master nuovo*)
	VAR_MNM_OutCvrAlarm : BOOL; (*1.6*)
	VAR_MNM_InCvrFixSpeedLimit : BOOL; (*V1.61*) (*Master nuovo*)
	VAR_MNM_InCvrFixSpeed : REAL; (*1.6*) (*Master nuovo*)
	VAR_MNM_OutCvrFixSpeedLimit : BOOL; (*V1.61*)
	VAR_MNM_OutCvrFixSpeed : REAL; (*1.6*)
	VAR_MNM_InCvrRampDwStart : REAL; (*V1.61*) (*Master nuovo*)
	VAR_MNM_OutCvrRampDwStart : REAL; (*V1.61*)
	TMR_TON_MNM_InCvrFix : TON; (*1.6*) (*Master nuovo*)
	TMR_TON_MNM_InCvrRamp : TON; (*1.6*) (*Master nuovo*)
	TMR_TON_MNM_OutCvrFix : TON; (*1.6*)
	TMR_TON_MNM_OutCvrRamp : TON; (*1.6*)
END_VAR
(*Speed Manager*)
VAR
	iSpeed : USINT;
	VAR_FixSpeed : ARRAY[1..CST_FixSpeedMax] OF VAR_FixSpeed_Type;
	VAR_FixSpeedActive : USINT;
	VAR_InFixSpeedActive : USINT;
	VAR_FlrFixSpeedActive : USINT;
	VAR_OutFixSpeedActive : USINT;
	VAR_ModuleSpeed : VAR_ModuleSpeed_Type;
END_VAR
VAR CONSTANT
	CST_FixSpeedMax : USINT := 15;
END_VAR
VAR
	TON_ReachedDelay : ARRAY[1..CST_FixSpeedMax] OF TON;
	VAR_MNM_FixSpeedReq : BOOL;
	VAR_MNM_FlrFixSpeedReq : BOOL;
	VAR_MNM_OutFixSpeedReq : BOOL;
	VAR_MNM_InFixSpeedReq : BOOL;
	TON_ContainerInletSafety1 : TON; (*V4.A.A.1.7.0*)
END_VAR
(*Master MNM Version*)
VAR
	VAR_MNM_version : INT := 100; (*v4.a.a.1.7.0 only for internal use*)
END_VAR
(*VAR TEST FOR DBA*)
VAR
	VAR_MNM_PccTestReversePos : INT; (*v999*)
	VAR_MNM_PccTestSecondHalf : INT; (*v999*)
	VAR_MNM_PccTestFirstHalf : INT; (*v999*)
END_VAR
```
